// TwinCAT 3 PLC project PLC_TMO_VAC
// ProgramVersion: 3.1.4022.7
// libraries:
//   LCLS General, * (SLAC)
//   LCLS Vacuum, * (SLAC - LCLS)
//   LCLSVacuumSerialDriverLib, * (SLAC - LCLS)
//   PMPS, * (SLAC - LCLS)
//   Tc2_SerialCom, * (Beckhoff Automation GmbH)
//   Tc2_Standard, * (Beckhoff Automation GmbH)
//   Tc2_System, * (Beckhoff Automation GmbH)
//   Tc3_Module, * (Beckhoff Automation GmbH)
// project tree:
//   / ComTask.TcTTO (not stored), FSVTask.TcTTO (not stored), PlcTask.TcTTO (not stored)
//   GVLs/ GVL_COM.TcGVL (not stored), GVL_FEE_Device.TcGVL, GVL_FSV_PMPS.TcGVL, GVL_FS_Devices.TcGVL, GVL_Hutch_Gauges.TcGVL, GVL_Hutch_Pumps.TcGVL (not stored), GVL_Hutch_Valves.TcGVL (not stored), GVL_PMPS.TcGVL, GVL_Variables.TcGVL
//   POUs/ DIAGNOSTICS.TcPOU, F_Turbo_Protection_ILK.TcPOU (not stored), MAIN.TcPOU, PMPS.TcPOU, PRG_COM.TcPOU (not stored), PRG_FEE.TcPOU, PRG_FSV.TcPOU, PRG_FSV_Interfaces.TcPOU (not stored), PRG_Hutch_Beamline_Valves.TcPOU (not stored), PRG_Hutch_Gauges.TcPOU (not stored), PRG_Roughing_Pumps.TcPOU, PRG_Section_2.TcPOU (not stored)
// real-time tasks:
//   TASK PlcTask: cycle T#10ms, priority 20, ADS port 350
//   TASK ComTask: cycle T#11ms, priority 1, ADS port 351
//   TASK FSVTask: cycle T#2ms, priority 2, ADS port 352
// I/O:
//   DEVICE Device 1 (EtherCAT), AmsNetId 172.21.132.22.2.1
//     B940-R20-CX0 (EK1200) [EK1200-5000 EtherCAT Power supply (2A E-Bus)]
//       CX0_E1 (EL2202)
//       CX0_E2_EXILK (EL1008)
//       CX0_E3 (EL2008)
//       CX0_E4 (EL2794)
//       CX0_E5 (EL6070)
//       CX0_E6_QPC1 (EL3064)
//       CX0_E7_QPC1 (EL1004)
//       CX0_E8_QPC1 (EL2794)
//       CX0_E9_QPC2 (EL3064)
//       CX0_E10_QPC2 (EL1004)
//       CX0_E11_QPC2 (EL2794)
//       CX0_E12 (EL6001)
//       EK1122-0080
//       PMPS_PRE
//       CX0_EK1110
//     B940_R20_EK0 (EK1100) [EK1100 EtherCAT Coupler (2A E-Bus)]
//       R20_EK0_E1 (EL3064)
//       R20_EK0_E2 (EL3064)
//       R20_EK0_E3 (EL2794)
//       R20_EK0_E4 (EL9505)
//       R20_EK0_E5 (EL1124)
//       R20_EK0_E6 (EK1110)
//     B940_K4S20_EK0  (EK1100)
//     B940_K4S20_EB1  (EP2338-0002)
//     B940_K4S20_EB2  (EP3174-0002)
//     B940_K4S20_EB3 (EP2624-0002)
//     B940_K4S24_EB1 (EP3174-0002)
//     B940_K4S24_EB2 (EP2624-0002)
//     B940_K4S28_EB1 (EP3174-0002)
//     B940_K4S28_EB2 (EP2624-0002)
//     B940_K4S33_EB1 (EP2338-0002)
//     B940_K4S33_EB2 (EP3174-0002)
//     B940_K4S33_EB3 (EP2624-0002)
//     TMO_WALL_WEST_EP01 (EP4374-0002)
//     TMO_K4S2_DRL_01 (EK1100)
//     TMO_K4S2_DRL_02 (EK1100)
//     TMO_K4S2_ EP1 (EP4374-0002)
//     TMO_K4S6_ EP1 (EP4374-0002)
//     TMO_K4S6_DRL_01 (EK1100)
//     TMO_K4S8_DRL_01 (EK1100)
// variable links:
//   PLC_TMO_VAC Instance <-> Device 1 (EtherCAT)/B940-R20-CX0 (EK1200)/CX0_E1 (EL2202)
//     PlcTask Outputs/GVL_PMPS.g_FastFaultOutput1.q_xFastFaultOut <-> Channel 1/Output
//     PlcTask Outputs/GVL_PMPS.g_FastFaultOutput2.q_xFastFaultOut <-> Channel 2/Output
//   PLC_TMO_VAC Instance <-> Device 1 (EtherCAT)/B940-R20-CX0 (EK1200)/CX0_E10_QPC2 (EL1004)
//     PlcTask Inputs/GVL_FEE_Device.PC4K4_XTES_PIP_01.i_xSP_DI <-> Channel 1/Input
//     PlcTask Inputs/GVL_Hutch_Pumps.MR2K4_KBO_PIP_01.i_xSP_DI <-> Channel 2/Input
//     PlcTask Inputs/GVL_Hutch_Pumps.MR4K4_KBO_PIP_01.i_xSP_DI <-> Channel 4/Input
//     PlcTask Inputs/GVL_Hutch_Pumps.PA2K4_IP1_PIP_01.i_xSP_DI <-> Channel 3/Input
//   PLC_TMO_VAC Instance <-> Device 1 (EtherCAT)/B940-R20-CX0 (EK1200)/CX0_E11_QPC2 (EL2794)
//     PlcTask Outputs/GVL_FEE_Device.PC4K4_XTES_PIP_01.q_xHVEna_DO <-> Channel 1/Output
//     PlcTask Outputs/GVL_Hutch_Pumps.MR2K4_KBO_PIP_01.q_xHVEna_DO <-> Channel 2/Output
//     PlcTask Outputs/GVL_Hutch_Pumps.MR4K4_KBO_PIP_01.q_xHVEna_DO <-> Channel 4/Output
//     PlcTask Outputs/GVL_Hutch_Pumps.PA2K4_IP1_PIP_01.q_xHVEna_DO <-> Channel 3/Output
//   PLC_TMO_VAC Instance <-> Device 1 (EtherCAT)/B940-R20-CX0 (EK1200)/CX0_E2_EXILK (EL1008)
//     PlcTask Inputs/GVL_FEE_Device.USVacOk_HI <-> Channel 1/Input
//     PlcTask Inputs/GVL_FEE_Device.USVacOk_LO <-> Channel 3/Input
//   PLC_TMO_VAC Instance <-> Device 1 (EtherCAT)/B940-R20-CX0 (EK1200)/CX0_E6_QPC1 (EL3064)
//     PlcTask Inputs/GVL_FEE_Device.MR1K4_SOMS_PIP_01.i_iPRESS <-> AI Standard Channel 1/Value
//     PlcTask Inputs/GVL_FEE_Device.ST1K4_TEST_PIP_01.i_iPRESS <-> AI Standard Channel 2/Value
//     PlcTask Inputs/GVL_FEE_Device.ST2K4_BCS_PIP_01.i_iPRESS <-> AI Standard Channel 3/Value
//     PlcTask Inputs/GVL_FEE_Device.ST3K4_PPS_PIP_01.i_iPRESS <-> AI Standard Channel 4/Value
//   PLC_TMO_VAC Instance <-> Device 1 (EtherCAT)/B940-R20-CX0 (EK1200)/CX0_E7_QPC1 (EL1004)
//     PlcTask Inputs/GVL_FEE_Device.MR1K4_SOMS_PIP_01.i_xSP_DI <-> Channel 1/Input
//     PlcTask Inputs/GVL_FEE_Device.ST1K4_TEST_PIP_01.i_xSP_DI <-> Channel 2/Input
//     PlcTask Inputs/GVL_FEE_Device.ST2K4_BCS_PIP_01.i_xSP_DI <-> Channel 3/Input
//     PlcTask Inputs/GVL_FEE_Device.ST3K4_PPS_PIP_01.i_xSP_DI <-> Channel 4/Input
//   PLC_TMO_VAC Instance <-> Device 1 (EtherCAT)/B940-R20-CX0 (EK1200)/CX0_E8_QPC1 (EL2794)
//     PlcTask Outputs/GVL_FEE_Device.MR1K4_SOMS_PIP_01.q_xHVEna_DO <-> Channel 1/Output
//     PlcTask Outputs/GVL_FEE_Device.ST1K4_TEST_PIP_01.q_xHVEna_DO <-> Channel 2/Output
//     PlcTask Outputs/GVL_FEE_Device.ST2K4_BCS_PIP_01.q_xHVEna_DO <-> Channel 3/Output
//     PlcTask Outputs/GVL_FEE_Device.ST3K4_PPS_PIP_01.q_xHVEna_DO <-> Channel 4/Output
//   PLC_TMO_VAC Instance <-> Device 1 (EtherCAT)/B940-R20-CX0 (EK1200)/CX0_E9_QPC2 (EL3064)
//     PlcTask Inputs/GVL_FEE_Device.PC4K4_XTES_PIP_01.i_iPRESS <-> AI Standard Channel 1/Value
//     PlcTask Inputs/GVL_Hutch_Pumps.MR2K4_KBO_PIP_01.i_iPRESS <-> AI Standard Channel 2/Value
//     PlcTask Inputs/GVL_Hutch_Pumps.MR4K4_KBO_PIP_01.i_iPRESS <-> AI Standard Channel 4/Value
//     PlcTask Inputs/GVL_Hutch_Pumps.PA2K4_IP1_PIP_01.i_iPRESS <-> AI Standard Channel 3/Value
//   PLC_TMO_VAC Instance <-> Device 1 (EtherCAT)/B940-R20-CX0 (EK1200)/PMPS_PRE
//     PlcTask Inputs/PMPS.fbArbiterIO.i_stCurrentBP <-> IO Inputs/CurrentBP
//     PlcTask Inputs/PMPS.fbArbiterIO.xTxPDO_state <-> SYNC Inputs/TxPDO state
//     PlcTask Inputs/PMPS.fbArbiterIO.xTxPDO_toggle <-> SYNC Inputs/TxPDO toggle
//     PlcTask Outputs/PMPS.fbArbiterIO.q_stRequestedBP <-> IO Outputs/RequestedBP
//   PLC_TMO_VAC Instance <-> Device 1 (EtherCAT)/B940_K4S20_EB1  (EP2338-0002)
//     PlcTask Inputs/GVL_FEE_Device.TV1K4_VGC_01.i_xClsLS <-> Channel 2/Input
//     PlcTask Inputs/GVL_FEE_Device.TV1K4_VGC_02.i_xClsLS <-> Channel 6/Input
//     PlcTask Inputs/GVL_FEE_Device.TV1K4_VGC_01.i_xOpnLS <-> Channel 1/Input
//     PlcTask Inputs/GVL_FEE_Device.TV1K4_VGC_02.i_xOpnLS <-> Channel 5/Input
//     PlcTask Outputs/GVL_FEE_Device.TV1K4_VGC_01.q_xOPN_DO <-> Channel 11/Output
//     PlcTask Outputs/GVL_FEE_Device.TV1K4_VGC_02.q_xOPN_DO <-> Channel 15/Output
//   PLC_TMO_VAC Instance <-> Device 1 (EtherCAT)/B940_K4S20_EB2  (EP3174-0002)
//     PlcTask Inputs/GVL_FEE_Device.TV1K4_GCC_01.i_iPRESS_R <-> AI Standard Channel 2/Value
//     PlcTask Inputs/GVL_FEE_Device.TV1K4_GPI_01.i_iPRESS_R <-> AI Standard Channel 1/Value
//   PLC_TMO_VAC Instance <-> Device 1 (EtherCAT)/B940_K4S20_EB3 (EP2624-0002)
//     PlcTask Outputs/GVL_FEE_Device.TV1K4_GCC_01.q_xHV_DIS <-> Channel 1/Output
//   PLC_TMO_VAC Instance <-> Device 1 (EtherCAT)/B940_K4S24_EB1 (EP3174-0002)
//     PlcTask Inputs/GVL_FEE_Device.ST1K4_TEST_GCC_01.i_iPRESS_R <-> AI Standard Channel 2/Value
//     PlcTask Inputs/GVL_FEE_Device.ST1K4_TEST_GPI_01.i_iPRESS_R <-> AI Standard Channel 1/Value
//   PLC_TMO_VAC Instance <-> Device 1 (EtherCAT)/B940_K4S24_EB2 (EP2624-0002)
//     PlcTask Outputs/GVL_FEE_Device.ST1K4_TEST_GCC_01.q_xHV_DIS <-> Channel 1/Output
//   PLC_TMO_VAC Instance <-> Device 1 (EtherCAT)/B940_K4S28_EB1 (EP3174-0002)
//     PlcTask Inputs/GVL_FEE_Device.ST2K4_BCS_GCC_01.i_iPRESS_R <-> AI Standard Channel 2/Value
//     PlcTask Inputs/GVL_FEE_Device.ST2K4_BCS_GPI_01.i_iPRESS_R <-> AI Standard Channel 1/Value
//   PLC_TMO_VAC Instance <-> Device 1 (EtherCAT)/B940_K4S28_EB2 (EP2624-0002)
//     PlcTask Outputs/GVL_FEE_Device.ST2K4_BCS_GCC_01.q_xHV_DIS <-> Channel 1/Output
//   PLC_TMO_VAC Instance <-> Device 1 (EtherCAT)/B940_K4S33_EB1 (EP2338-0002)
//     PlcTask Inputs/GVL_FEE_Device.ST3K4_PPS_VGC_01.i_xClsLS <-> Channel 2/Input
//     PlcTask Inputs/GVL_FEE_Device.ST3K4_PPS_VGC_01.i_xOpnLS <-> Channel 1/Input
//     PlcTask Outputs/GVL_FEE_Device.ST3K4_PPS_VGC_01.q_xOPN_DO <-> Channel 11/Output
//   PLC_TMO_VAC Instance <-> Device 1 (EtherCAT)/B940_K4S33_EB2 (EP3174-0002)
//     PlcTask Inputs/GVL_FEE_Device.PC4K4_XTES_GCC_01.i_iPRESS_R <-> AI Standard Channel 2/Value
//     PlcTask Inputs/GVL_FEE_Device.PC4K4_XTES_GPI_01.i_iPRESS_R <-> AI Standard Channel 1/Value
//   PLC_TMO_VAC Instance <-> Device 1 (EtherCAT)/B940_K4S33_EB3 (EP2624-0002)
//     PlcTask Outputs/GVL_FEE_Device.PC4K4_XTES_GCC_01.q_xHV_DIS <-> Channel 1/Output
//   PLC_TMO_VAC Instance <-> Device 1 (EtherCAT)/B940_R20_EK0 (EK1100)/R20_EK0_E5_MKS937B (EL1124)
//     FSVTask Inputs/GVL_FS_Devices.MR3K4_KBO_VFS_1.i_xTrigger <-> Channel 1/Input
//     FSVTask Inputs/GVL_FS_Devices.MR4K4_KBO_VFS_1.i_xTrigger <-> Channel 1/Input
//     FSVTask Inputs/GVL_FS_Devices.TV1K4_VFS_1.i_xTrigger <-> Channel 1/Input
//   PLC_TMO_VAC Instance <-> Device 1 (EtherCAT)/TMO_K4S2_ EP1 (EP4374-0002)
//     PlcTask Inputs/GVL_Hutch_Gauges.TMO_ROUGH1_GPI_02.i_iPRESS_R <-> AI Inputs Channel 1/Value
//     PlcTask Inputs/GVL_Hutch_Gauges.TMO_ROUGH2_GPI_02.i_iPRESS_R <-> AI Inputs Channel 2/Value
//     PlcTask Outputs/GVL_Hutch_Valves.TMO_ROUGH1_VFV_02.q_iRawPosition <-> AO Outputs Channel 3/Analog output
//     PlcTask Outputs/GVL_Hutch_Valves.TMO_ROUGH2_VFV_01.q_iRawPosition <-> AO Outputs Channel 4/Analog output
//   PLC_TMO_VAC Instance <-> Device 1 (EtherCAT)/TMO_K4S2_DRL_01 (EK1100)/K4S2_01_E1_VFS (EL1004)
//     FSVTask Inputs/GVL_FS_Devices.MR3K4_KBO_VFS_1.i_xClsLS <-> Channel 1/Input
//     FSVTask Inputs/GVL_FS_Devices.MR3K4_KBO_VFS_1.i_xOpnLS <-> Channel 2/Input
//   PLC_TMO_VAC Instance <-> Device 1 (EtherCAT)/TMO_K4S2_DRL_01 (EK1100)/K4S2_01_E3_VFS (EL2202)
//     FSVTask Outputs/GVL_FS_Devices.MR3K4_KBO_VFS_1.q_xClose_A <-> Channel 1/Output
//     FSVTask Outputs/GVL_FS_Devices.MR3K4_KBO_VFS_1.q_xClose_B <-> Channel 2/Output
//   PLC_TMO_VAC Instance <-> Device 1 (EtherCAT)/TMO_K4S2_DRL_01 (EK1100)/K4S2_01_E4_VFS (EL2202)
//     FSVTask Outputs/GVL_FS_Devices.MR3K4_KBO_VFS_1.q_xClose_C <-> Channel 1/Output
//     FSVTask Outputs/GVL_FS_Devices.MR3K4_KBO_VFS_1.q_xOPN_DO <-> Channel 2/Output
//   PLC_TMO_VAC Instance <-> Device 1 (EtherCAT)/TMO_K4S2_DRL_01 (EK1100)/K4S2_01_E5 (EL1004)
//     PlcTask Inputs/GVL_Hutch_Valves.MR2K4_KBO_VWC_01.i_xClsLS <-> Channel 2/Input
//     PlcTask Inputs/GVL_Hutch_Valves.MR3K4_KBO_VWC_01.i_xClsLS <-> Channel 4/Input
//     PlcTask Inputs/GVL_Hutch_Valves.MR2K4_KBO_VWC_01.i_xOpnLS <-> Channel 1/Input
//     PlcTask Inputs/GVL_Hutch_Valves.MR3K4_KBO_VWC_01.i_xOpnLS <-> Channel 3/Input
//   PLC_TMO_VAC Instance <-> Device 1 (EtherCAT)/TMO_K4S2_DRL_01 (EK1100)/K4S2_01_E6 (EL2004)
//     PlcTask Outputs/GVL_Hutch_Valves.MR2K4_KBO_VWC_01.q_xOPN_DO <-> Channel 1/Output
//     PlcTask Outputs/GVL_Hutch_Valves.MR3K4_KBO_VWC_01.q_xOPN_DO <-> Channel 2/Output
//   PLC_TMO_VAC Instance <-> Device 1 (EtherCAT)/TMO_K4S2_DRL_02 (EK1100)/K4S2_02_E1 (EL3174)
//     PlcTask Inputs/GVL_Hutch_Gauges.MR2K4_KBO_GCC_01.i_iPRESS_R <-> AI Standard Channel 3/Value
//     PlcTask Inputs/GVL_Hutch_Gauges.MR2K4_KBO_GPI_01.i_iPRESS_R <-> AI Standard Channel 2/Value
//     PlcTask Inputs/GVL_Hutch_Gauges.PA1K4_IP1_GCC_01.i_iPRESS_R <-> AI Standard Channel 4/Value
//   PLC_TMO_VAC Instance <-> Device 1 (EtherCAT)/TMO_K4S2_DRL_02 (EK1100)/K4S2_02_E10 (EL6021)
//     ComTask Inputs/GVL_COM.K4S2_02_E10_stComIn/D[0] <-> COM TxPDO-Map Inputs/Data In 0
//     ComTask Inputs/GVL_COM.K4S2_02_E10_stComIn/D[10] <-> COM TxPDO-Map Inputs/Data In 10
//     ComTask Inputs/GVL_COM.K4S2_02_E10_stComIn/D[11] <-> COM TxPDO-Map Inputs/Data In 11
//     ComTask Inputs/GVL_COM.K4S2_02_E10_stComIn/D[12] <-> COM TxPDO-Map Inputs/Data In 12
//     ComTask Inputs/GVL_COM.K4S2_02_E10_stComIn/D[13] <-> COM TxPDO-Map Inputs/Data In 13
//     ComTask Inputs/GVL_COM.K4S2_02_E10_stComIn/D[14] <-> COM TxPDO-Map Inputs/Data In 14
//     ComTask Inputs/GVL_COM.K4S2_02_E10_stComIn/D[15] <-> COM TxPDO-Map Inputs/Data In 15
//     ComTask Inputs/GVL_COM.K4S2_02_E10_stComIn/D[16] <-> COM TxPDO-Map Inputs/Data In 16
//     ComTask Inputs/GVL_COM.K4S2_02_E10_stComIn/D[17] <-> COM TxPDO-Map Inputs/Data In 17
//     ComTask Inputs/GVL_COM.K4S2_02_E10_stComIn/D[18] <-> COM TxPDO-Map Inputs/Data In 18
//     ComTask Inputs/GVL_COM.K4S2_02_E10_stComIn/D[19] <-> COM TxPDO-Map Inputs/Data In 19
//     ComTask Inputs/GVL_COM.K4S2_02_E10_stComIn/D[1] <-> COM TxPDO-Map Inputs/Data In 1
//     ComTask Inputs/GVL_COM.K4S2_02_E10_stComIn/D[20] <-> COM TxPDO-Map Inputs/Data In 20
//     ComTask Inputs/GVL_COM.K4S2_02_E10_stComIn/D[21] <-> COM TxPDO-Map Inputs/Data In 21
//     ComTask Inputs/GVL_COM.K4S2_02_E10_stComIn/D[2] <-> COM TxPDO-Map Inputs/Data In 2
//     ComTask Inputs/GVL_COM.K4S2_02_E10_stComIn/D[3] <-> COM TxPDO-Map Inputs/Data In 3
//     ComTask Inputs/GVL_COM.K4S2_02_E10_stComIn/D[4] <-> COM TxPDO-Map Inputs/Data In 4
//     ComTask Inputs/GVL_COM.K4S2_02_E10_stComIn/D[5] <-> COM TxPDO-Map Inputs/Data In 5
//     ComTask Inputs/GVL_COM.K4S2_02_E10_stComIn/D[6] <-> COM TxPDO-Map Inputs/Data In 6
//     ComTask Inputs/GVL_COM.K4S2_02_E10_stComIn/D[7] <-> COM TxPDO-Map Inputs/Data In 7
//     ComTask Inputs/GVL_COM.K4S2_02_E10_stComIn/D[8] <-> COM TxPDO-Map Inputs/Data In 8
//     ComTask Inputs/GVL_COM.K4S2_02_E10_stComIn/D[9] <-> COM TxPDO-Map Inputs/Data In 9
//     ComTask Inputs/GVL_COM.K4S2_02_E10_stComIn/Status <-> COM TxPDO-Map Inputs/Status
//     ComTask Outputs/GVL_COM.K4S2_02_E10_stComOut/Ctrl <-> COM RxPDO-Map Outputs/Ctrl
//     ComTask Outputs/GVL_COM.K4S2_02_E10_stComOut/D[0] <-> COM RxPDO-Map Outputs/Data Out 0
//     ComTask Outputs/GVL_COM.K4S2_02_E10_stComOut/D[10] <-> COM RxPDO-Map Outputs/Data Out 10
//     ComTask Outputs/GVL_COM.K4S2_02_E10_stComOut/D[11] <-> COM RxPDO-Map Outputs/Data Out 11
//     ComTask Outputs/GVL_COM.K4S2_02_E10_stComOut/D[12] <-> COM RxPDO-Map Outputs/Data Out 12
//     ComTask Outputs/GVL_COM.K4S2_02_E10_stComOut/D[13] <-> COM RxPDO-Map Outputs/Data Out 13
//     ComTask Outputs/GVL_COM.K4S2_02_E10_stComOut/D[14] <-> COM RxPDO-Map Outputs/Data Out 14
//     ComTask Outputs/GVL_COM.K4S2_02_E10_stComOut/D[15] <-> COM RxPDO-Map Outputs/Data Out 15
//     ComTask Outputs/GVL_COM.K4S2_02_E10_stComOut/D[16] <-> COM RxPDO-Map Outputs/Data Out 16
//     ComTask Outputs/GVL_COM.K4S2_02_E10_stComOut/D[17] <-> COM RxPDO-Map Outputs/Data Out 17
//     ComTask Outputs/GVL_COM.K4S2_02_E10_stComOut/D[18] <-> COM RxPDO-Map Outputs/Data Out 18
//     ComTask Outputs/GVL_COM.K4S2_02_E10_stComOut/D[19] <-> COM RxPDO-Map Outputs/Data Out 19
//     ComTask Outputs/GVL_COM.K4S2_02_E10_stComOut/D[1] <-> COM RxPDO-Map Outputs/Data Out 1
//     ComTask Outputs/GVL_COM.K4S2_02_E10_stComOut/D[20] <-> COM RxPDO-Map Outputs/Data Out 20
//     ComTask Outputs/GVL_COM.K4S2_02_E10_stComOut/D[21] <-> COM RxPDO-Map Outputs/Data Out 21
//     ComTask Outputs/GVL_COM.K4S2_02_E10_stComOut/D[2] <-> COM RxPDO-Map Outputs/Data Out 2
//     ComTask Outputs/GVL_COM.K4S2_02_E10_stComOut/D[3] <-> COM RxPDO-Map Outputs/Data Out 3
//     ComTask Outputs/GVL_COM.K4S2_02_E10_stComOut/D[4] <-> COM RxPDO-Map Outputs/Data Out 4
//     ComTask Outputs/GVL_COM.K4S2_02_E10_stComOut/D[5] <-> COM RxPDO-Map Outputs/Data Out 5
//     ComTask Outputs/GVL_COM.K4S2_02_E10_stComOut/D[6] <-> COM RxPDO-Map Outputs/Data Out 6
//     ComTask Outputs/GVL_COM.K4S2_02_E10_stComOut/D[7] <-> COM RxPDO-Map Outputs/Data Out 7
//     ComTask Outputs/GVL_COM.K4S2_02_E10_stComOut/D[8] <-> COM RxPDO-Map Outputs/Data Out 8
//     ComTask Outputs/GVL_COM.K4S2_02_E10_stComOut/D[9] <-> COM RxPDO-Map Outputs/Data Out 9
//   PLC_TMO_VAC Instance <-> Device 1 (EtherCAT)/TMO_K4S2_DRL_02 (EK1100)/K4S2_02_E11 (EL1004)
//     PlcTask Inputs/GVL_Hutch_Pumps.PA1K4_IP1_PTM_01.i_xAtSpd <-> Channel 2/Input
//     PlcTask Inputs/GVL_Hutch_Pumps.PA1K4_IP1_PTM_02.i_xAtSpd <-> Channel 4/Input
//     PlcTask Inputs/GVL_Hutch_Pumps.PA1K4_IP1_PTM_01.i_xFaultNC <-> Channel 1/Input
//     PlcTask Inputs/GVL_Hutch_Pumps.PA1K4_IP1_PTM_02.i_xFaultNC <-> Channel 3/Input
//   PLC_TMO_VAC Instance <-> Device 1 (EtherCAT)/TMO_K4S2_DRL_02 (EK1100)/K4S2_02_E12 (EL2794)
//     PlcTask Outputs/GVL_Hutch_Pumps.PA1K4_IP1_PTM_01.q_RunDO <-> Channel 1/Output
//     PlcTask Outputs/GVL_Hutch_Pumps.PA1K4_IP1_PTM_02.q_RunDO <-> Channel 3/Output
//     PlcTask Outputs/GVL_Hutch_Pumps.PA1K4_IP1_PTM_01.q_xReset <-> Channel 2/Output
//     PlcTask Outputs/GVL_Hutch_Pumps.PA1K4_IP1_PTM_02.q_xReset <-> Channel 4/Output
//   PLC_TMO_VAC Instance <-> Device 1 (EtherCAT)/TMO_K4S2_DRL_02 (EK1100)/K4S2_02_E13 (EL1004)
//     PlcTask Inputs/GVL_Hutch_Pumps.PA1K4_IP1_PTM_03.i_xAtSpd <-> Channel 2/Input
//     PlcTask Inputs/GVL_Hutch_Pumps.PA1K4_IP1_PTM_03.i_xFaultNC <-> Channel 1/Input
//   PLC_TMO_VAC Instance <-> Device 1 (EtherCAT)/TMO_K4S2_DRL_02 (EK1100)/K4S2_02_E14 (EL2794)
//     PlcTask Outputs/GVL_Hutch_Pumps.PA1K4_IP1_PTM_03.q_RunDO <-> Channel 1/Output
//     PlcTask Outputs/GVL_Hutch_Pumps.PA1K4_IP1_PTM_03.q_xReset <-> Channel 2/Output
//   PLC_TMO_VAC Instance <-> Device 1 (EtherCAT)/TMO_K4S2_DRL_02 (EK1100)/K4S2_02_E15 (EL1004)
//     PlcTask Inputs/GVL_Hutch_Pumps.IM4K4_PPM_PTM_01.i_xAtSpd <-> Channel 2/Input
//     PlcTask Inputs/GVL_Hutch_Pumps.IM4K4_PPM_PTM_01.i_xFaultNC <-> Channel 1/Input
//     PlcTask Inputs/GVL_Hutch_Pumps.LI1K4_IP1_PTM_01.i_xAtSpd <-> Channel 4/Input
//     PlcTask Inputs/GVL_Hutch_Pumps.LI1K4_IP1_PTM_01.i_xFaultNC <-> Channel 3/Input
//   PLC_TMO_VAC Instance <-> Device 1 (EtherCAT)/TMO_K4S2_DRL_02 (EK1100)/K4S2_02_E16 (EL2794)
//     PlcTask Outputs/GVL_Hutch_Pumps.IM4K4_PPM_PTM_01.q_RunDO <-> Channel 1/Output
//     PlcTask Outputs/GVL_Hutch_Pumps.LI1K4_IP1_PTM_01.q_RunDO <-> Channel 2/Output
//   PLC_TMO_VAC Instance <-> Device 1 (EtherCAT)/TMO_K4S2_DRL_02 (EK1100)/K4S2_02_E17 (EL6001)
//     ComTask Inputs/GVL_COM.K4S2_02_E17_stComIn/D[0] <-> COM Inputs/Data In 0
//     ComTask Inputs/GVL_COM.K4S2_02_E17_stComIn/D[10] <-> COM Inputs/Data In 10
//     ComTask Inputs/GVL_COM.K4S2_02_E17_stComIn/D[11] <-> COM Inputs/Data In 11
//     ComTask Inputs/GVL_COM.K4S2_02_E17_stComIn/D[12] <-> COM Inputs/Data In 12
//     ComTask Inputs/GVL_COM.K4S2_02_E17_stComIn/D[13] <-> COM Inputs/Data In 13
//     ComTask Inputs/GVL_COM.K4S2_02_E17_stComIn/D[14] <-> COM Inputs/Data In 14
//     ComTask Inputs/GVL_COM.K4S2_02_E17_stComIn/D[15] <-> COM Inputs/Data In 15
//     ComTask Inputs/GVL_COM.K4S2_02_E17_stComIn/D[16] <-> COM Inputs/Data In 16
//     ComTask Inputs/GVL_COM.K4S2_02_E17_stComIn/D[17] <-> COM Inputs/Data In 17
//     ComTask Inputs/GVL_COM.K4S2_02_E17_stComIn/D[18] <-> COM Inputs/Data In 18
//     ComTask Inputs/GVL_COM.K4S2_02_E17_stComIn/D[19] <-> COM Inputs/Data In 19
//     ComTask Inputs/GVL_COM.K4S2_02_E17_stComIn/D[1] <-> COM Inputs/Data In 1
//     ComTask Inputs/GVL_COM.K4S2_02_E17_stComIn/D[20] <-> COM Inputs/Data In 20
//     ComTask Inputs/GVL_COM.K4S2_02_E17_stComIn/D[21] <-> COM Inputs/Data In 21
//     ComTask Inputs/GVL_COM.K4S2_02_E17_stComIn/D[2] <-> COM Inputs/Data In 2
//     ComTask Inputs/GVL_COM.K4S2_02_E17_stComIn/D[3] <-> COM Inputs/Data In 3
//     ComTask Inputs/GVL_COM.K4S2_02_E17_stComIn/D[4] <-> COM Inputs/Data In 4
//     ComTask Inputs/GVL_COM.K4S2_02_E17_stComIn/D[5] <-> COM Inputs/Data In 5
//     ComTask Inputs/GVL_COM.K4S2_02_E17_stComIn/D[6] <-> COM Inputs/Data In 6
//     ComTask Inputs/GVL_COM.K4S2_02_E17_stComIn/D[7] <-> COM Inputs/Data In 7
//     ComTask Inputs/GVL_COM.K4S2_02_E17_stComIn/D[8] <-> COM Inputs/Data In 8
//     ComTask Inputs/GVL_COM.K4S2_02_E17_stComIn/D[9] <-> COM Inputs/Data In 9
//     ComTask Inputs/GVL_COM.K4S2_02_E17_stComIn/Status <-> COM Inputs/Status
//     ComTask Outputs/GVL_COM.K4S2_02_E17_stComOut/Ctrl <-> COM Outputs/Ctrl
//     ComTask Outputs/GVL_COM.K4S2_02_E17_stComOut/D[0] <-> COM Outputs/Data Out 0
//     ComTask Outputs/GVL_COM.K4S2_02_E17_stComOut/D[10] <-> COM Outputs/Data Out 10
//     ComTask Outputs/GVL_COM.K4S2_02_E17_stComOut/D[11] <-> COM Outputs/Data Out 11
//     ComTask Outputs/GVL_COM.K4S2_02_E17_stComOut/D[12] <-> COM Outputs/Data Out 12
//     ComTask Outputs/GVL_COM.K4S2_02_E17_stComOut/D[13] <-> COM Outputs/Data Out 13
//     ComTask Outputs/GVL_COM.K4S2_02_E17_stComOut/D[14] <-> COM Outputs/Data Out 14
//     ComTask Outputs/GVL_COM.K4S2_02_E17_stComOut/D[15] <-> COM Outputs/Data Out 15
//     ComTask Outputs/GVL_COM.K4S2_02_E17_stComOut/D[16] <-> COM Outputs/Data Out 16
//     ComTask Outputs/GVL_COM.K4S2_02_E17_stComOut/D[17] <-> COM Outputs/Data Out 17
//     ComTask Outputs/GVL_COM.K4S2_02_E17_stComOut/D[18] <-> COM Outputs/Data Out 18
//     ComTask Outputs/GVL_COM.K4S2_02_E17_stComOut/D[19] <-> COM Outputs/Data Out 19
//     ComTask Outputs/GVL_COM.K4S2_02_E17_stComOut/D[1] <-> COM Outputs/Data Out 1
//     ComTask Outputs/GVL_COM.K4S2_02_E17_stComOut/D[20] <-> COM Outputs/Data Out 20
//     ComTask Outputs/GVL_COM.K4S2_02_E17_stComOut/D[21] <-> COM Outputs/Data Out 21
//     ComTask Outputs/GVL_COM.K4S2_02_E17_stComOut/D[2] <-> COM Outputs/Data Out 2
//     ComTask Outputs/GVL_COM.K4S2_02_E17_stComOut/D[3] <-> COM Outputs/Data Out 3
//     ComTask Outputs/GVL_COM.K4S2_02_E17_stComOut/D[4] <-> COM Outputs/Data Out 4
//     ComTask Outputs/GVL_COM.K4S2_02_E17_stComOut/D[5] <-> COM Outputs/Data Out 5
//     ComTask Outputs/GVL_COM.K4S2_02_E17_stComOut/D[6] <-> COM Outputs/Data Out 6
//     ComTask Outputs/GVL_COM.K4S2_02_E17_stComOut/D[7] <-> COM Outputs/Data Out 7
//     ComTask Outputs/GVL_COM.K4S2_02_E17_stComOut/D[8] <-> COM Outputs/Data Out 8
//     ComTask Outputs/GVL_COM.K4S2_02_E17_stComOut/D[9] <-> COM Outputs/Data Out 9
//   PLC_TMO_VAC Instance <-> Device 1 (EtherCAT)/TMO_K4S2_DRL_02 (EK1100)/K4S2_02_E18 (EL6001)
//     ComTask Inputs/GVL_COM.K4S2_02_E18_stComIn/D[0] <-> COM Inputs/Data In 0
//     ComTask Inputs/GVL_COM.K4S2_02_E18_stComIn/D[10] <-> COM Inputs/Data In 10
//     ComTask Inputs/GVL_COM.K4S2_02_E18_stComIn/D[11] <-> COM Inputs/Data In 11
//     ComTask Inputs/GVL_COM.K4S2_02_E18_stComIn/D[12] <-> COM Inputs/Data In 12
//     ComTask Inputs/GVL_COM.K4S2_02_E18_stComIn/D[13] <-> COM Inputs/Data In 13
//     ComTask Inputs/GVL_COM.K4S2_02_E18_stComIn/D[14] <-> COM Inputs/Data In 14
//     ComTask Inputs/GVL_COM.K4S2_02_E18_stComIn/D[15] <-> COM Inputs/Data In 15
//     ComTask Inputs/GVL_COM.K4S2_02_E18_stComIn/D[16] <-> COM Inputs/Data In 16
//     ComTask Inputs/GVL_COM.K4S2_02_E18_stComIn/D[17] <-> COM Inputs/Data In 17
//     ComTask Inputs/GVL_COM.K4S2_02_E18_stComIn/D[18] <-> COM Inputs/Data In 18
//     ComTask Inputs/GVL_COM.K4S2_02_E18_stComIn/D[19] <-> COM Inputs/Data In 19
//     ComTask Inputs/GVL_COM.K4S2_02_E18_stComIn/D[1] <-> COM Inputs/Data In 1
//     ComTask Inputs/GVL_COM.K4S2_02_E18_stComIn/D[20] <-> COM Inputs/Data In 20
//     ComTask Inputs/GVL_COM.K4S2_02_E18_stComIn/D[21] <-> COM Inputs/Data In 21
//     ComTask Inputs/GVL_COM.K4S2_02_E18_stComIn/D[2] <-> COM Inputs/Data In 2
//     ComTask Inputs/GVL_COM.K4S2_02_E18_stComIn/D[3] <-> COM Inputs/Data In 3
//     ComTask Inputs/GVL_COM.K4S2_02_E18_stComIn/D[4] <-> COM Inputs/Data In 4
//     ComTask Inputs/GVL_COM.K4S2_02_E18_stComIn/D[5] <-> COM Inputs/Data In 5
//     ComTask Inputs/GVL_COM.K4S2_02_E18_stComIn/D[6] <-> COM Inputs/Data In 6
//     ComTask Inputs/GVL_COM.K4S2_02_E18_stComIn/D[7] <-> COM Inputs/Data In 7
//     ComTask Inputs/GVL_COM.K4S2_02_E18_stComIn/D[8] <-> COM Inputs/Data In 8
//     ComTask Inputs/GVL_COM.K4S2_02_E18_stComIn/D[9] <-> COM Inputs/Data In 9
//     ComTask Inputs/GVL_COM.K4S2_02_E18_stComIn/Status <-> COM Inputs/Status
//     ComTask Outputs/GVL_COM.K4S2_02_E18_stComOut/Ctrl <-> COM Outputs/Ctrl
//     ComTask Outputs/GVL_COM.K4S2_02_E18_stComOut/D[0] <-> COM Outputs/Data Out 0
//     ComTask Outputs/GVL_COM.K4S2_02_E18_stComOut/D[10] <-> COM Outputs/Data Out 10
//     ComTask Outputs/GVL_COM.K4S2_02_E18_stComOut/D[11] <-> COM Outputs/Data Out 11
//     ComTask Outputs/GVL_COM.K4S2_02_E18_stComOut/D[12] <-> COM Outputs/Data Out 12
//     ComTask Outputs/GVL_COM.K4S2_02_E18_stComOut/D[13] <-> COM Outputs/Data Out 13
//     ComTask Outputs/GVL_COM.K4S2_02_E18_stComOut/D[14] <-> COM Outputs/Data Out 14
//     ComTask Outputs/GVL_COM.K4S2_02_E18_stComOut/D[15] <-> COM Outputs/Data Out 15
//     ComTask Outputs/GVL_COM.K4S2_02_E18_stComOut/D[16] <-> COM Outputs/Data Out 16
//     ComTask Outputs/GVL_COM.K4S2_02_E18_stComOut/D[17] <-> COM Outputs/Data Out 17
//     ComTask Outputs/GVL_COM.K4S2_02_E18_stComOut/D[18] <-> COM Outputs/Data Out 18
//     ComTask Outputs/GVL_COM.K4S2_02_E18_stComOut/D[19] <-> COM Outputs/Data Out 19
//     ComTask Outputs/GVL_COM.K4S2_02_E18_stComOut/D[1] <-> COM Outputs/Data Out 1
//     ComTask Outputs/GVL_COM.K4S2_02_E18_stComOut/D[20] <-> COM Outputs/Data Out 20
//     ComTask Outputs/GVL_COM.K4S2_02_E18_stComOut/D[21] <-> COM Outputs/Data Out 21
//     ComTask Outputs/GVL_COM.K4S2_02_E18_stComOut/D[2] <-> COM Outputs/Data Out 2
//     ComTask Outputs/GVL_COM.K4S2_02_E18_stComOut/D[3] <-> COM Outputs/Data Out 3
//     ComTask Outputs/GVL_COM.K4S2_02_E18_stComOut/D[4] <-> COM Outputs/Data Out 4
//     ComTask Outputs/GVL_COM.K4S2_02_E18_stComOut/D[5] <-> COM Outputs/Data Out 5
//     ComTask Outputs/GVL_COM.K4S2_02_E18_stComOut/D[6] <-> COM Outputs/Data Out 6
//     ComTask Outputs/GVL_COM.K4S2_02_E18_stComOut/D[7] <-> COM Outputs/Data Out 7
//     ComTask Outputs/GVL_COM.K4S2_02_E18_stComOut/D[8] <-> COM Outputs/Data Out 8
//     ComTask Outputs/GVL_COM.K4S2_02_E18_stComOut/D[9] <-> COM Outputs/Data Out 9
//   PLC_TMO_VAC Instance <-> Device 1 (EtherCAT)/TMO_K4S2_DRL_02 (EK1100)/K4S2_02_E19 (EL1004)
//     PlcTask Inputs/GVL_Hutch_Valves.TMO_ROUGH1_VRC_01.i_xClsLS <-> Channel 2/Input
//     PlcTask Inputs/GVL_Hutch_Valves.TMO_ROUGH2_VRC_01.i_xClsLS <-> Channel 4/Input
//     PlcTask Inputs/GVL_Hutch_Valves.TMO_ROUGH1_VRC_01.i_xOpnLS <-> Channel 1/Input
//     PlcTask Inputs/GVL_Hutch_Valves.TMO_ROUGH2_VRC_01.i_xOpnLS <-> Channel 3/Input
//   PLC_TMO_VAC Instance <-> Device 1 (EtherCAT)/TMO_K4S2_DRL_02 (EK1100)/K4S2_02_E2 (EL3174)
//     PlcTask Inputs/GVL_Hutch_Gauges.IM4K4_PPM_GCC_01.i_iPRESS_R <-> AI Standard Channel 2/Value
//     PlcTask Inputs/GVL_Hutch_Gauges.PA1K4_IP1_GPI_01.i_iPRESS_R <-> AI Standard Channel 1/Value
//   PLC_TMO_VAC Instance <-> Device 1 (EtherCAT)/TMO_K4S2_DRL_02 (EK1100)/K4S2_02_E20 (EL2004)
//     PlcTask Outputs/GVL_Hutch_Valves.TMO_ROUGH1_VRC_01.q_xOPN_DO <-> Channel 1/Output
//     PlcTask Outputs/GVL_Hutch_Valves.TMO_ROUGH2_VRC_01.q_xOPN_DO <-> Channel 2/Output
//   PLC_TMO_VAC Instance <-> Device 1 (EtherCAT)/TMO_K4S2_DRL_02 (EK1100)/K4S2_02_E5 (EL2624)
//     PlcTask Outputs/GVL_Hutch_Gauges.IM4K4_PPM_GCC_01.q_xHV_DIS <-> Channel 4/Output
//     PlcTask Outputs/GVL_Hutch_Gauges.MR2K4_KBO_GCC_01.q_xHV_DIS <-> Channel 2/Output
//     PlcTask Outputs/GVL_Hutch_Gauges.PA1K4_IP1_GCC_01.q_xHV_DIS <-> Channel 3/Output
//   PLC_TMO_VAC Instance <-> Device 1 (EtherCAT)/TMO_K4S2_DRL_02 (EK1100)/K4S2_02_E7 (EL1124)
//     PlcTask Inputs/GVL_Hutch_Gauges.MR2K4_KBO_GCC_01.i_xDisc_Active <-> Channel 4/Input
//     PlcTask Inputs/GVL_Hutch_Gauges.MR2K4_KBO_GCC_01.i_xHV_ON <-> Channel 3/Input
//   PLC_TMO_VAC Instance <-> Device 1 (EtherCAT)/TMO_K4S2_DRL_02 (EK1100)/K4S2_02_E8 (EL1124)
//     PlcTask Inputs/GVL_Hutch_Gauges.IM4K4_PPM_GCC_01.i_xDisc_Active <-> Channel 4/Input
//     PlcTask Inputs/GVL_Hutch_Gauges.IM4K4_PPM_GCC_01.i_xHV_ON <-> Channel 3/Input
//     PlcTask Inputs/GVL_Hutch_Gauges.PA1K4_IP1_GCC_01.i_xDisc_Active <-> Channel 2/Input
//     PlcTask Inputs/GVL_Hutch_Gauges.PA1K4_IP1_GCC_01.i_xHV_ON <-> Channel 1/Input
//   PLC_TMO_VAC Instance <-> Device 1 (EtherCAT)/TMO_K4S6_ EP1 (EP4374-0002)
//     PlcTask Inputs/GVL_Hutch_Gauges.TMO_ROUGH1_GPI_03.i_iPRESS_R <-> AI Inputs Channel 1/Value
//     PlcTask Outputs/GVL_Hutch_Valves.TMO_ROUGH1_VFV_03.q_iRawPosition <-> AO Outputs Channel 3/Analog output
//   PLC_TMO_VAC Instance <-> Device 1 (EtherCAT)/TMO_K4S6_DRL_01 (EK1100)/K4S6_01_E1 (EL1004)
//     PlcTask Inputs/GVL_Hutch_Valves.TMO_ROUGH1_VRC_02.i_xClsLS <-> Channel 2/Input
//     PlcTask Inputs/GVL_Hutch_Valves.TMO_ROUGH1_VRC_02.i_xOpnLS <-> Channel 1/Input
//   PLC_TMO_VAC Instance <-> Device 1 (EtherCAT)/TMO_K4S6_DRL_01 (EK1100)/K4S6_01_E11 (EL1004)
//     PlcTask Inputs/GVL_Hutch_Pumps.IM5K4_PPM_PTM_01.i_xFaultNC <-> Channel 1/Input
//   PLC_TMO_VAC Instance <-> Device 1 (EtherCAT)/TMO_K4S6_DRL_01 (EK1100)/K4S6_01_E12 (EL2004)
//     PlcTask Outputs/GVL_Hutch_Pumps.IM5K4_PPM_PTM_01.q_PumpingStation <-> Channel 1/Output
//   PLC_TMO_VAC Instance <-> Device 1 (EtherCAT)/TMO_K4S6_DRL_01 (EK1100)/K4S6_01_E14 (EL2624)
//     PlcTask Outputs/GVL_Hutch_Gauges.IM5K4_PPM_GCC_01.q_xHV_DIS <-> Channel 2/Output
//     PlcTask Outputs/GVL_Hutch_Gauges.MR4K4_KBO_GCC_01.q_xHV_DIS <-> Channel 4/Output
//     PlcTask Outputs/GVL_Hutch_Gauges.PA2K4_IP1_GCC_01.q_xHV_DIS <-> Channel 3/Output
//     PlcTask Outputs/GVL_Hutch_Gauges.TM1K4_GCC_01.q_xHV_DIS <-> Channel 1/Output
//   PLC_TMO_VAC Instance <-> Device 1 (EtherCAT)/TMO_K4S6_DRL_01 (EK1100)/K4S6_01_E15 (EL3174)
//     PlcTask Inputs/GVL_Hutch_Gauges.IM5K4_PPM_GCC_01.i_iPRESS_R <-> AI Standard Channel 2/Value
//     PlcTask Inputs/GVL_Hutch_Gauges.PA2K4_IP1_GCC_01.i_iPRESS_R <-> AI Standard Channel 3/Value
//     PlcTask Inputs/GVL_Hutch_Gauges.PA2K4_IP1_GPI_01.i_iPRESS_R <-> AI Standard Channel 4/Value
//     PlcTask Inputs/GVL_Hutch_Gauges.TM1K4_GCC_01.i_iPRESS_R <-> AI Standard Channel 1/Value
//   PLC_TMO_VAC Instance <-> Device 1 (EtherCAT)/TMO_K4S6_DRL_01 (EK1100)/K4S6_01_E18 (EL3174)
//     PlcTask Inputs/GVL_Hutch_Gauges.MR4K4_KBO_GCC_01.i_iPRESS_R <-> AI Standard Channel 2/Value
//     PlcTask Inputs/GVL_Hutch_Gauges.MR4K4_KBO_GPI_01.i_iPRESS_R <-> AI Standard Channel 1/Value
//   PLC_TMO_VAC Instance <-> Device 1 (EtherCAT)/TMO_K4S6_DRL_01 (EK1100)/K4S6_01_E2 (EL2004)
//     PlcTask Outputs/GVL_Hutch_Valves.TMO_ROUGH1_VRC_02.q_xOPN_DO <-> Channel 1/Output
//   PLC_TMO_VAC Instance <-> Device 1 (EtherCAT)/TMO_K4S6_DRL_01 (EK1100)/K4S6_01_E20 (EL1124)
//     PlcTask Inputs/GVL_Hutch_Gauges.IM5K4_PPM_GCC_01.i_xDisc_Active <-> Channel 4/Input
//     PlcTask Inputs/GVL_Hutch_Gauges.IM5K4_PPM_GCC_01.i_xHV_ON <-> Channel 3/Input
//     PlcTask Inputs/GVL_Hutch_Gauges.TM1K4_GCC_01.i_xDisc_Active <-> Channel 2/Input
//     PlcTask Inputs/GVL_Hutch_Gauges.TM1K4_GCC_01.i_xHV_ON <-> Channel 1/Input
//   PLC_TMO_VAC Instance <-> Device 1 (EtherCAT)/TMO_K4S6_DRL_01 (EK1100)/K4S6_01_E21 (EL1124)
//     PlcTask Inputs/GVL_Hutch_Gauges.MR4K4_KBO_GCC_01.i_xDisc_Active <-> Channel 4/Input
//     PlcTask Inputs/GVL_Hutch_Gauges.MR4K4_KBO_GCC_01.i_xHV_ON <-> Channel 3/Input
//     PlcTask Inputs/GVL_Hutch_Gauges.PA2K4_IP1_GCC_01.i_xDisc_Active <-> Channel 2/Input
//     PlcTask Inputs/GVL_Hutch_Gauges.PA2K4_IP1_GCC_01.i_xHV_ON <-> Channel 1/Input
//   PLC_TMO_VAC Instance <-> Device 1 (EtherCAT)/TMO_K4S6_DRL_01 (EK1100)/K4S6_01_E22_IP1 (EL1004)
//     PlcTask Inputs/GVL_Variables.xLAMP_PTM_NOK <-> Channel 1/Input
//   PLC_TMO_VAC Instance <-> Device 1 (EtherCAT)/TMO_K4S6_DRL_01 (EK1100)/K4S6_01_E3 (EL1004)
//     PlcTask Inputs/GVL_Hutch_Valves.LI3K4_IP1_VWC_01.i_xClsLS <-> Channel 2/Input
//     PlcTask Inputs/GVL_Hutch_Valves.LI3K4_IP1_VWC_01.i_xOpnLS <-> Channel 1/Input
//     PlcTask Inputs/GVL_Hutch_Valves.PC5K4_VWC_01.i_xClsLS <-> Channel 4/Input
//     PlcTask Inputs/GVL_Hutch_Valves.PC5K4_VWC_01.i_xOpnLS <-> Channel 3/Input
//   PLC_TMO_VAC Instance <-> Device 1 (EtherCAT)/TMO_K4S6_DRL_01 (EK1100)/K4S6_01_E4 (EL2004)
//     PlcTask Outputs/GVL_Hutch_Valves.LI3K4_IP1_VWC_01.q_xOPN_DO <-> Channel 1/Output
//     PlcTask Outputs/GVL_Hutch_Valves.PC5K4_VWC_01.q_xOPN_DO <-> Channel 2/Output
//   PLC_TMO_VAC Instance <-> Device 1 (EtherCAT)/TMO_K4S6_DRL_01 (EK1100)/K4S6_01_E5 (EL6021)
//     ComTask Inputs/GVL_COM.K4S6_01_E5_stComIn/D[0] <-> COM TxPDO-Map Inputs/Data In 0
//     ComTask Inputs/GVL_COM.K4S6_01_E5_stComIn/D[10] <-> COM TxPDO-Map Inputs/Data In 10
//     ComTask Inputs/GVL_COM.K4S6_01_E5_stComIn/D[11] <-> COM TxPDO-Map Inputs/Data In 11
//     ComTask Inputs/GVL_COM.K4S6_01_E5_stComIn/D[12] <-> COM TxPDO-Map Inputs/Data In 12
//     ComTask Inputs/GVL_COM.K4S6_01_E5_stComIn/D[13] <-> COM TxPDO-Map Inputs/Data In 13
//     ComTask Inputs/GVL_COM.K4S6_01_E5_stComIn/D[14] <-> COM TxPDO-Map Inputs/Data In 14
//     ComTask Inputs/GVL_COM.K4S6_01_E5_stComIn/D[15] <-> COM TxPDO-Map Inputs/Data In 15
//     ComTask Inputs/GVL_COM.K4S6_01_E5_stComIn/D[16] <-> COM TxPDO-Map Inputs/Data In 16
//     ComTask Inputs/GVL_COM.K4S6_01_E5_stComIn/D[17] <-> COM TxPDO-Map Inputs/Data In 17
//     ComTask Inputs/GVL_COM.K4S6_01_E5_stComIn/D[18] <-> COM TxPDO-Map Inputs/Data In 18
//     ComTask Inputs/GVL_COM.K4S6_01_E5_stComIn/D[19] <-> COM TxPDO-Map Inputs/Data In 19
//     ComTask Inputs/GVL_COM.K4S6_01_E5_stComIn/D[1] <-> COM TxPDO-Map Inputs/Data In 1
//     ComTask Inputs/GVL_COM.K4S6_01_E5_stComIn/D[20] <-> COM TxPDO-Map Inputs/Data In 20
//     ComTask Inputs/GVL_COM.K4S6_01_E5_stComIn/D[21] <-> COM TxPDO-Map Inputs/Data In 21
//     ComTask Inputs/GVL_COM.K4S6_01_E5_stComIn/D[2] <-> COM TxPDO-Map Inputs/Data In 2
//     ComTask Inputs/GVL_COM.K4S6_01_E5_stComIn/D[3] <-> COM TxPDO-Map Inputs/Data In 3
//     ComTask Inputs/GVL_COM.K4S6_01_E5_stComIn/D[4] <-> COM TxPDO-Map Inputs/Data In 4
//     ComTask Inputs/GVL_COM.K4S6_01_E5_stComIn/D[5] <-> COM TxPDO-Map Inputs/Data In 5
//     ComTask Inputs/GVL_COM.K4S6_01_E5_stComIn/D[6] <-> COM TxPDO-Map Inputs/Data In 6
//     ComTask Inputs/GVL_COM.K4S6_01_E5_stComIn/D[7] <-> COM TxPDO-Map Inputs/Data In 7
//     ComTask Inputs/GVL_COM.K4S6_01_E5_stComIn/D[8] <-> COM TxPDO-Map Inputs/Data In 8
//     ComTask Inputs/GVL_COM.K4S6_01_E5_stComIn/D[9] <-> COM TxPDO-Map Inputs/Data In 9
//     ComTask Inputs/GVL_COM.K4S6_01_E5_stComIn/Status <-> COM TxPDO-Map Inputs/Status
//     ComTask Outputs/GVL_COM.K4S6_01_E5_stComOut/Ctrl <-> COM RxPDO-Map Outputs/Ctrl
//     ComTask Outputs/GVL_COM.K4S6_01_E5_stComOut/D[0] <-> COM RxPDO-Map Outputs/Data Out 0
//     ComTask Outputs/GVL_COM.K4S6_01_E5_stComOut/D[10] <-> COM RxPDO-Map Outputs/Data Out 10
//     ComTask Outputs/GVL_COM.K4S6_01_E5_stComOut/D[11] <-> COM RxPDO-Map Outputs/Data Out 11
//     ComTask Outputs/GVL_COM.K4S6_01_E5_stComOut/D[12] <-> COM RxPDO-Map Outputs/Data Out 12
//     ComTask Outputs/GVL_COM.K4S6_01_E5_stComOut/D[13] <-> COM RxPDO-Map Outputs/Data Out 13
//     ComTask Outputs/GVL_COM.K4S6_01_E5_stComOut/D[14] <-> COM RxPDO-Map Outputs/Data Out 14
//     ComTask Outputs/GVL_COM.K4S6_01_E5_stComOut/D[15] <-> COM RxPDO-Map Outputs/Data Out 15
//     ComTask Outputs/GVL_COM.K4S6_01_E5_stComOut/D[16] <-> COM RxPDO-Map Outputs/Data Out 16
//     ComTask Outputs/GVL_COM.K4S6_01_E5_stComOut/D[17] <-> COM RxPDO-Map Outputs/Data Out 17
//     ComTask Outputs/GVL_COM.K4S6_01_E5_stComOut/D[18] <-> COM RxPDO-Map Outputs/Data Out 18
//     ComTask Outputs/GVL_COM.K4S6_01_E5_stComOut/D[19] <-> COM RxPDO-Map Outputs/Data Out 19
//     ComTask Outputs/GVL_COM.K4S6_01_E5_stComOut/D[1] <-> COM RxPDO-Map Outputs/Data Out 1
//     ComTask Outputs/GVL_COM.K4S6_01_E5_stComOut/D[20] <-> COM RxPDO-Map Outputs/Data Out 20
//     ComTask Outputs/GVL_COM.K4S6_01_E5_stComOut/D[21] <-> COM RxPDO-Map Outputs/Data Out 21
//     ComTask Outputs/GVL_COM.K4S6_01_E5_stComOut/D[2] <-> COM RxPDO-Map Outputs/Data Out 2
//     ComTask Outputs/GVL_COM.K4S6_01_E5_stComOut/D[3] <-> COM RxPDO-Map Outputs/Data Out 3
//     ComTask Outputs/GVL_COM.K4S6_01_E5_stComOut/D[4] <-> COM RxPDO-Map Outputs/Data Out 4
//     ComTask Outputs/GVL_COM.K4S6_01_E5_stComOut/D[5] <-> COM RxPDO-Map Outputs/Data Out 5
//     ComTask Outputs/GVL_COM.K4S6_01_E5_stComOut/D[6] <-> COM RxPDO-Map Outputs/Data Out 6
//     ComTask Outputs/GVL_COM.K4S6_01_E5_stComOut/D[7] <-> COM RxPDO-Map Outputs/Data Out 7
//     ComTask Outputs/GVL_COM.K4S6_01_E5_stComOut/D[8] <-> COM RxPDO-Map Outputs/Data Out 8
//     ComTask Outputs/GVL_COM.K4S6_01_E5_stComOut/D[9] <-> COM RxPDO-Map Outputs/Data Out 9
//   PLC_TMO_VAC Instance <-> Device 1 (EtherCAT)/TMO_K4S6_DRL_01 (EK1100)/K4S6_01_E6 (EL1004)
//     PlcTask Inputs/GVL_Hutch_Pumps.LI3K4_IP1_OUT_PTM_01.i_xAtSpd <-> Channel 1/Input
//     PlcTask Inputs/GVL_Hutch_Pumps.LI3K4_IP1_OUT_PTM_01.i_xFaultNC <-> Channel 3/Input
//     PlcTask Inputs/GVL_Hutch_Pumps.LI3K4_IP1_OUT_PTM_01.i_xRemote <-> Channel 2/Input
//     PlcTask Inputs/GVL_Hutch_Pumps.TM1K4_PTM_01.i_xAtSpd <-> Channel 4/Input
//   PLC_TMO_VAC Instance <-> Device 1 (EtherCAT)/TMO_K4S6_DRL_01 (EK1100)/K4S6_01_E7 (EL2004)
//     PlcTask Outputs/GVL_Hutch_Pumps.LI3K4_IP1_OUT_PTM_01.q_PumpingStation <-> Channel 3/Output
//     PlcTask Outputs/GVL_Hutch_Pumps.LI3K4_IP1_OUT_PTM_01.q_RunDO <-> Channel 1/Output
//     PlcTask Outputs/GVL_Hutch_Pumps.LI3K4_IP1_OUT_PTM_01.q_xRemote <-> Channel 2/Output
//     PlcTask Outputs/GVL_Hutch_Pumps.TM1K4_PTM_01.q_RunDO <-> Channel 4/Output
//   PLC_TMO_VAC Instance <-> Device 1 (EtherCAT)/TMO_K4S6_DRL_01 (EK1100)/K4S6_01_E8 (EL1004)
//     PlcTask Inputs/GVL_Hutch_Pumps.IM5K4_PPM_PTM_01.i_xAtSpd <-> Channel 3/Input
//     PlcTask Inputs/GVL_Hutch_Pumps.IM5K4_PPM_PTM_01.i_xRemote <-> Channel 4/Input
//     PlcTask Inputs/GVL_Hutch_Pumps.TM1K4_PTM_01.i_xFaultNC <-> Channel 2/Input
//     PlcTask Inputs/GVL_Hutch_Pumps.TM1K4_PTM_01.i_xRemote <-> Channel 1/Input
//   PLC_TMO_VAC Instance <-> Device 1 (EtherCAT)/TMO_K4S6_DRL_01 (EK1100)/K4S6_01_E9 (EL2004)
//     PlcTask Outputs/GVL_Hutch_Pumps.IM5K4_PPM_PTM_01.q_RunDO <-> Channel 3/Output
//     PlcTask Outputs/GVL_Hutch_Pumps.IM5K4_PPM_PTM_01.q_xRemote <-> Channel 4/Output
//     PlcTask Outputs/GVL_Hutch_Pumps.TM1K4_PTM_01.q_PumpingStation <-> Channel 2/Output
//     PlcTask Outputs/GVL_Hutch_Pumps.TM1K4_PTM_01.q_xRemote <-> Channel 1/Output
//   PLC_TMO_VAC Instance <-> Device 1 (EtherCAT)/TMO_K4S8_DRL_01 (EK1100)/K4S8_01_E1 (EL1004)
//     FSVTask Inputs/GVL_FS_Devices.MR4K4_KBO_VFS_1.i_xClsLS <-> Channel 1/Input
//     FSVTask Inputs/GVL_FS_Devices.MR4K4_KBO_VFS_1.i_xOpnLS <-> Channel 2/Input
//   PLC_TMO_VAC Instance <-> Device 1 (EtherCAT)/TMO_K4S8_DRL_01 (EK1100)/K4S8_01_E3 (EL2202)
//     FSVTask Outputs/GVL_FS_Devices.MR4K4_KBO_VFS_1.q_xClose_A <-> Channel 1/Output
//     FSVTask Outputs/GVL_FS_Devices.MR4K4_KBO_VFS_1.q_xClose_B <-> Channel 2/Output
//   PLC_TMO_VAC Instance <-> Device 1 (EtherCAT)/TMO_K4S8_DRL_01 (EK1100)/K4S8_01_E4 (EL2202)
//     FSVTask Outputs/GVL_FS_Devices.MR4K4_KBO_VFS_1.q_xClose_C <-> Channel 1/Output
//     FSVTask Outputs/GVL_FS_Devices.MR4K4_KBO_VFS_1.q_xOPN_DO <-> Channel 2/Output
//   PLC_TMO_VAC Instance <-> Device 1 (EtherCAT)/TMO_K4S8_DRL_01 (EK1100)/K4S8_01_E5 (EL1004)
//     PlcTask Inputs/GVL_Hutch_Valves.MR4K4_KBO_VWC_01.i_xClsLS <-> Channel 2/Input
//     PlcTask Inputs/GVL_Hutch_Valves.MR5K4_KBO_VWC_01.i_xClsLS <-> Channel 4/Input
//     PlcTask Inputs/GVL_Hutch_Valves.MR4K4_KBO_VWC_01.i_xOpnLS <-> Channel 1/Input
//     PlcTask Inputs/GVL_Hutch_Valves.MR5K4_KBO_VWC_01.i_xOpnLS <-> Channel 3/Input
//   PLC_TMO_VAC Instance <-> Device 1 (EtherCAT)/TMO_K4S8_DRL_01 (EK1100)/K4S8_01_E6 (EL2004)
//     PlcTask Outputs/GVL_Hutch_Valves.MR4K4_KBO_VWC_01.q_xOPN_DO <-> Channel 1/Output
//     PlcTask Outputs/GVL_Hutch_Valves.MR5K4_KBO_VWC_01.q_xOPN_DO <-> Channel 2/Output
//   PLC_TMO_VAC Instance <-> Device 1 (EtherCAT)/TMO_WALL_WEST_EP01 (EP4374-0002)
//     PlcTask Inputs/GVL_Hutch_Gauges.TMO_ROUGH1_GPI_01.i_iPRESS_R <-> AI Inputs Channel 1/Value
//     PlcTask Inputs/GVL_Hutch_Gauges.TMO_ROUGH2_GPI_01.i_iPRESS_R <-> AI Inputs Channel 2/Value
//     PlcTask Outputs/GVL_Hutch_Valves.TMO_ROUGH1_VFV_01.q_iRawPosition <-> AO Outputs Channel 3/Analog output
//   PLC_TMO_VAC Instance <-> PLC_TMO_VAC/PLC_TMO_VAC Instance
//     FSVTask Inputs/GVL_FS_Devices.MR3K4_KBO_VFS_1.i_xCLS_SW <-> PlcTask Outputs/GVL_FS_Devices.MR3K4_KBO_VFS_Interface.q_xCLS_SW
//     FSVTask Inputs/GVL_FS_Devices.MR4K4_KBO_VFS_1.i_xCLS_SW <-> PlcTask Outputs/GVL_FS_Devices.MR4K4_KBO_VFS_Interface.q_xCLS_SW
//     FSVTask Inputs/GVL_FS_Devices.MR3K4_KBO_VFS_1.i_xOPN_SW <-> PlcTask Outputs/GVL_FS_Devices.MR3K4_KBO_VFS_Interface.q_xOPN_SW
//     FSVTask Inputs/GVL_FS_Devices.MR4K4_KBO_VFS_1.i_xOPN_SW <-> PlcTask Outputs/GVL_FS_Devices.MR4K4_KBO_VFS_Interface.q_xOPN_SW
//     FSVTask Inputs/GVL_FS_Devices.MR3K4_KBO_VFS_1.i_xOverrideMode <-> PlcTask Outputs/GVL_FS_Devices.MR3K4_KBO_VFS_Interface.q_xOverrideMode
//     FSVTask Inputs/GVL_FS_Devices.MR4K4_KBO_VFS_1.i_xOverrideMode <-> PlcTask Outputs/GVL_FS_Devices.MR4K4_KBO_VFS_Interface.q_xOverrideMode
//     FSVTask Inputs/GVL_FS_Devices.MR3K4_KBO_VFS_1.i_xOverrideOpen <-> PlcTask Outputs/GVL_FS_Devices.MR3K4_KBO_VFS_Interface.q_xOverrideOpen
//     FSVTask Inputs/GVL_FS_Devices.MR4K4_KBO_VFS_1.i_xOverrideOpen <-> PlcTask Outputs/GVL_FS_Devices.MR4K4_KBO_VFS_Interface.q_xOverrideOpen
//     FSVTask Inputs/GVL_FS_Devices.MR3K4_KBO_VFS_1.i_xPress_OK <-> PlcTask Outputs/GVL_FS_Devices.MR3K4_KBO_VFS_Interface.q_xPRESS_OK
//     FSVTask Inputs/GVL_FS_Devices.MR4K4_KBO_VFS_1.i_xPress_OK <-> PlcTask Outputs/GVL_FS_Devices.MR4K4_KBO_VFS_Interface.q_xPRESS_OK
//     FSVTask Inputs/GVL_FS_Devices.MR3K4_KBO_VFS_1.i_xVAC_FAULT_Reset <-> PlcTask Outputs/GVL_FS_Devices.MR3K4_KBO_VFS_Interface.q_xVAC_FAULT_Reset
//     FSVTask Inputs/GVL_FS_Devices.MR4K4_KBO_VFS_1.i_xVAC_FAULT_Reset <-> PlcTask Outputs/GVL_FS_Devices.MR4K4_KBO_VFS_Interface.q_xVAC_FAULT_Reset
//     FSVTask Inputs/GVL_FS_Devices.TV1K4_VFS_1.i_xCLS_SW <-> PlcTask Outputs/GVL_FS_Devices.TV1K4_VFS_Interface.q_xCLS_SW
//     FSVTask Inputs/GVL_FS_Devices.TV1K4_VFS_1.i_xOPN_SW <-> PlcTask Outputs/GVL_FS_Devices.TV1K4_VFS_Interface.q_xOPN_SW
//     FSVTask Inputs/GVL_FS_Devices.TV1K4_VFS_1.i_xOverrideMode <-> PlcTask Outputs/GVL_FS_Devices.TV1K4_VFS_Interface.q_xOverrideMode
//     FSVTask Inputs/GVL_FS_Devices.TV1K4_VFS_1.i_xOverrideOpen <-> PlcTask Outputs/GVL_FS_Devices.TV1K4_VFS_Interface.q_xOverrideOpen
//     FSVTask Inputs/GVL_FS_Devices.TV1K4_VFS_1.i_xPress_OK <-> PlcTask Outputs/GVL_FS_Devices.TV1K4_VFS_Interface.q_xPRESS_OK
//     FSVTask Inputs/GVL_FS_Devices.TV1K4_VFS_1.i_xVAC_FAULT_Reset <-> PlcTask Outputs/GVL_FS_Devices.TV1K4_VFS_Interface.q_xVAC_FAULT_Reset
//     FSVTask Outputs/GVL_FS_Devices.MR3K4_KBO_VFS_1.q_eVFS_State <-> PlcTask Inputs/GVL_FS_Devices.MR3K4_KBO_VFS_Interface.i_eVFS_State
//     FSVTask Outputs/GVL_FS_Devices.MR4K4_KBO_VFS_1.q_eVFS_State <-> PlcTask Inputs/GVL_FS_Devices.MR4K4_KBO_VFS_Interface.i_eVFS_State
//     FSVTask Outputs/GVL_FS_Devices.MR3K4_KBO_VFS_1.q_xMPS_OK <-> PlcTask Inputs/GVL_FS_Devices.MR3K4_KBO_VFS_Interface.i_xMPS_OK
//     FSVTask Outputs/GVL_FS_Devices.MR4K4_KBO_VFS_1.q_xMPS_OK <-> PlcTask Inputs/GVL_FS_Devices.MR4K4_KBO_VFS_Interface.i_xMPS_OK
//     FSVTask Outputs/GVL_FS_Devices.MR3K4_KBO_VFS_1.q_xVAC_FAULT_OK <-> PlcTask Inputs/GVL_FS_Devices.MR3K4_KBO_VFS_Interface.i_xVAC_FAULT_OK
//     FSVTask Outputs/GVL_FS_Devices.MR4K4_KBO_VFS_1.q_xVAC_FAULT_OK <-> PlcTask Inputs/GVL_FS_Devices.MR4K4_KBO_VFS_Interface.i_xVAC_FAULT_OK
//     FSVTask Outputs/GVL_FS_Devices.MR3K4_KBO_VFS_1.q_xVFS_Closed <-> PlcTask Inputs/GVL_FS_Devices.MR3K4_KBO_VFS_Interface.i_xVFS_Closed
//     FSVTask Outputs/GVL_FS_Devices.MR4K4_KBO_VFS_1.q_xVFS_Closed <-> PlcTask Inputs/GVL_FS_Devices.MR4K4_KBO_VFS_Interface.i_xVFS_Closed
//     FSVTask Outputs/GVL_FS_Devices.TV1K4_VFS_1.q_eVFS_State <-> PlcTask Inputs/GVL_FS_Devices.TV1K4_VFS_Interface.i_eVFS_State
//     FSVTask Outputs/GVL_FS_Devices.TV1K4_VFS_1.q_xMPS_OK <-> PlcTask Inputs/GVL_FS_Devices.TV1K4_VFS_Interface.i_xMPS_OK
//     FSVTask Outputs/GVL_FS_Devices.TV1K4_VFS_1.q_xVAC_FAULT_OK <-> PlcTask Inputs/GVL_FS_Devices.TV1K4_VFS_Interface.i_xVAC_FAULT_OK
//     FSVTask Outputs/GVL_FS_Devices.TV1K4_VFS_1.q_xVFS_Closed <-> PlcTask Inputs/GVL_FS_Devices.TV1K4_VFS_Interface.i_xVFS_Closed
//     PlcTask Inputs/GVL_FS_Devices.MR3K4_KBO_VFS_Interface.i_eVFS_State <-> FSVTask Outputs/GVL_FS_Devices.MR3K4_KBO_VFS_1.q_eVFS_State
//     PlcTask Inputs/GVL_FS_Devices.MR4K4_KBO_VFS_Interface.i_eVFS_State <-> FSVTask Outputs/GVL_FS_Devices.MR4K4_KBO_VFS_1.q_eVFS_State
//     PlcTask Inputs/GVL_FS_Devices.MR3K4_KBO_VFS_Interface.i_xMPS_OK <-> FSVTask Outputs/GVL_FS_Devices.MR3K4_KBO_VFS_1.q_xMPS_OK
//     PlcTask Inputs/GVL_FS_Devices.MR4K4_KBO_VFS_Interface.i_xMPS_OK <-> FSVTask Outputs/GVL_FS_Devices.MR4K4_KBO_VFS_1.q_xMPS_OK
//     PlcTask Inputs/GVL_FS_Devices.MR3K4_KBO_VFS_Interface.i_xVAC_FAULT_OK <-> FSVTask Outputs/GVL_FS_Devices.MR3K4_KBO_VFS_1.q_xVAC_FAULT_OK
//     PlcTask Inputs/GVL_FS_Devices.MR4K4_KBO_VFS_Interface.i_xVAC_FAULT_OK <-> FSVTask Outputs/GVL_FS_Devices.MR4K4_KBO_VFS_1.q_xVAC_FAULT_OK
//     PlcTask Inputs/GVL_FS_Devices.MR3K4_KBO_VFS_Interface.i_xVFS_Closed <-> FSVTask Outputs/GVL_FS_Devices.MR3K4_KBO_VFS_1.q_xVFS_Closed
//     PlcTask Inputs/GVL_FS_Devices.MR4K4_KBO_VFS_Interface.i_xVFS_Closed <-> FSVTask Outputs/GVL_FS_Devices.MR4K4_KBO_VFS_1.q_xVFS_Closed
//     PlcTask Inputs/GVL_FS_Devices.TV1K4_VFS_Interface.i_eVFS_State <-> FSVTask Outputs/GVL_FS_Devices.TV1K4_VFS_1.q_eVFS_State
//     PlcTask Inputs/GVL_FS_Devices.TV1K4_VFS_Interface.i_xMPS_OK <-> FSVTask Outputs/GVL_FS_Devices.TV1K4_VFS_1.q_xMPS_OK
//     PlcTask Inputs/GVL_FS_Devices.TV1K4_VFS_Interface.i_xVAC_FAULT_OK <-> FSVTask Outputs/GVL_FS_Devices.TV1K4_VFS_1.q_xVAC_FAULT_OK
//     PlcTask Inputs/GVL_FS_Devices.TV1K4_VFS_Interface.i_xVFS_Closed <-> FSVTask Outputs/GVL_FS_Devices.TV1K4_VFS_1.q_xVFS_Closed
//     PlcTask Outputs/GVL_FS_Devices.MR3K4_KBO_VFS_Interface.q_xCLS_SW <-> FSVTask Inputs/GVL_FS_Devices.MR3K4_KBO_VFS_1.i_xCLS_SW
//     PlcTask Outputs/GVL_FS_Devices.MR4K4_KBO_VFS_Interface.q_xCLS_SW <-> FSVTask Inputs/GVL_FS_Devices.MR4K4_KBO_VFS_1.i_xCLS_SW
//     PlcTask Outputs/GVL_FS_Devices.MR3K4_KBO_VFS_Interface.q_xOPN_SW <-> FSVTask Inputs/GVL_FS_Devices.MR3K4_KBO_VFS_1.i_xOPN_SW
//     PlcTask Outputs/GVL_FS_Devices.MR4K4_KBO_VFS_Interface.q_xOPN_SW <-> FSVTask Inputs/GVL_FS_Devices.MR4K4_KBO_VFS_1.i_xOPN_SW
//     PlcTask Outputs/GVL_FS_Devices.MR3K4_KBO_VFS_Interface.q_xOverrideMode <-> FSVTask Inputs/GVL_FS_Devices.MR3K4_KBO_VFS_1.i_xOverrideMode
//     PlcTask Outputs/GVL_FS_Devices.MR4K4_KBO_VFS_Interface.q_xOverrideMode <-> FSVTask Inputs/GVL_FS_Devices.MR4K4_KBO_VFS_1.i_xOverrideMode
//     PlcTask Outputs/GVL_FS_Devices.MR3K4_KBO_VFS_Interface.q_xOverrideOpen <-> FSVTask Inputs/GVL_FS_Devices.MR3K4_KBO_VFS_1.i_xOverrideOpen
//     PlcTask Outputs/GVL_FS_Devices.MR4K4_KBO_VFS_Interface.q_xOverrideOpen <-> FSVTask Inputs/GVL_FS_Devices.MR4K4_KBO_VFS_1.i_xOverrideOpen
//     PlcTask Outputs/GVL_FS_Devices.MR3K4_KBO_VFS_Interface.q_xPRESS_OK <-> FSVTask Inputs/GVL_FS_Devices.MR3K4_KBO_VFS_1.i_xPress_OK
//     PlcTask Outputs/GVL_FS_Devices.MR4K4_KBO_VFS_Interface.q_xPRESS_OK <-> FSVTask Inputs/GVL_FS_Devices.MR4K4_KBO_VFS_1.i_xPress_OK
//     PlcTask Outputs/GVL_FS_Devices.MR3K4_KBO_VFS_Interface.q_xVAC_FAULT_Reset <-> FSVTask Inputs/GVL_FS_Devices.MR3K4_KBO_VFS_1.i_xVAC_FAULT_Reset
//     PlcTask Outputs/GVL_FS_Devices.MR4K4_KBO_VFS_Interface.q_xVAC_FAULT_Reset <-> FSVTask Inputs/GVL_FS_Devices.MR4K4_KBO_VFS_1.i_xVAC_FAULT_Reset
//     PlcTask Outputs/GVL_FS_Devices.TV1K4_VFS_Interface.q_xCLS_SW <-> FSVTask Inputs/GVL_FS_Devices.TV1K4_VFS_1.i_xCLS_SW
//     PlcTask Outputs/GVL_FS_Devices.TV1K4_VFS_Interface.q_xOPN_SW <-> FSVTask Inputs/GVL_FS_Devices.TV1K4_VFS_1.i_xOPN_SW
//     PlcTask Outputs/GVL_FS_Devices.TV1K4_VFS_Interface.q_xOverrideMode <-> FSVTask Inputs/GVL_FS_Devices.TV1K4_VFS_1.i_xOverrideMode
//     PlcTask Outputs/GVL_FS_Devices.TV1K4_VFS_Interface.q_xOverrideOpen <-> FSVTask Inputs/GVL_FS_Devices.TV1K4_VFS_1.i_xOverrideOpen
//     PlcTask Outputs/GVL_FS_Devices.TV1K4_VFS_Interface.q_xPRESS_OK <-> FSVTask Inputs/GVL_FS_Devices.TV1K4_VFS_1.i_xPress_OK
//     PlcTask Outputs/GVL_FS_Devices.TV1K4_VFS_Interface.q_xVAC_FAULT_Reset <-> FSVTask Inputs/GVL_FS_Devices.TV1K4_VFS_1.i_xVAC_FAULT_Reset
//   PLC_TMO_VAC_FS Instance <-> Device 1 (EtherCAT)/B940_K4S20_EK0  (EK1100)/K4S20-E1-FSV (EL1004)
//     PlcTask Inputs/GVL_FS.TV1K4_VFS_01.i_xClsLS <-> Channel 1/Input
//     PlcTask Inputs/GVL_FS.TV1K4_VFS_01.i_xOpnLS <-> Channel 2/Input
//   PLC_TMO_VAC_FS Instance <-> Device 1 (EtherCAT)/B940_K4S20_EK0  (EK1100)/K4S20-E2-FSV (EL2202)
//     PlcTask Outputs/GVL_FS.TV1K4_VFS_01.q_xClose_A <-> Channel 1/Output
//     PlcTask Outputs/GVL_FS.TV1K4_VFS_01.q_xClose_B <-> Channel 2/Output
//   PLC_TMO_VAC_FS Instance <-> Device 1 (EtherCAT)/B940_K4S20_EK0  (EK1100)/K4S20-E3-FSV (EL2202)
//     PlcTask Outputs/GVL_FS.TV1K4_VFS_01.q_xClose_C <-> Channel 1/Output
//     PlcTask Outputs/GVL_FS.TV1K4_VFS_01.q_xOPN_DO <-> Channel 2/Output
//   PLC_TMO_VAC_FS Instance <-> Device 1 (EtherCAT)/B940_R20_EK0 (EK1100)/R20_EK0_E5 (EL1124)
//     PlcTask Inputs/GVL_FS.TV1K4_VFS_01.i_xTrigger <-> Channel 1/Input

// ---- GVLs/GVL_FEE_Device.TcGVL
//{attribute 'qualified_only'}
VAR_GLOBAL

(* upstream vacuum ok *)
   {attribute 'pytmc' :=' pv : USVAC:OK:HI '}
   {attribute 'TcLinkTo' := 	' := 	TIIB[CX0_E2_EXILK (EL1008)]^Channel 1^Input	'}	
   USVacOk_HI AT%I* : BOOL; (* upstream vacuum <10E-6, for mirror VGC interlock *)
 
 	{attribute 'pytmc' :=' pv : USVAC:OK:LO '}
   {attribute 'TcLinkTo' := 	'	:= 	TIIB[CX0_E2_EXILK (EL1008)]^Channel 3^Input	'}	  
   USVacOk_LO AT%I* : BOOL; (* upstream vacuum <10E-4, for Ion pump interlock *)


(* Isolation gate valves*)

	{attribute 'pytmc' :=' pv : TV1K4:VGC:01 '}
	{attribute 'TcLinkTo' := 	'.i_xOpnLS	:=	TIIB[B940_K4S20_EB1  (EP2338-0002)]^Channel 1^Input;
								 .i_xClsLS	:=	TIIB[B940_K4S20_EB1  (EP2338-0002)]^Channel 2^Input;
								.q_xOPN_DO	:=	TIIB[B940_K4S20_EB1  (EP2338-0002)]^Channel 11^Output'}
	TV1K4_VGC_01: FB_VGC;
	
	{attribute 'pytmc' :=' pv : TV1K4:VGC:02 '}
	{attribute 'TcLinkTo' := 	'.i_xOpnLS	:=	TIIB[B940_K4S20_EB1  (EP2338-0002)]^Channel 5^Input;
								 .i_xClsLS	:=	TIIB[B940_K4S20_EB1  (EP2338-0002)]^Channel 6^Input;
								 .q_xOPN_DO	:=	TIIB[B940_K4S20_EB1  (EP2338-0002)]^Channel 15^Output'}	
 	TV1K4_VGC_02: FB_VGC;

	{attribute 'pytmc' :=' pv : ST3K4:PPS:VGC:01 '}
	{attribute 'TcLinkTo' := 	'.i_xOpnLS	:=	TIIB[B940_K4S33_EB1 (EP2338-0002)]^Channel 1^Input;
								 .i_xClsLS	:=	TIIB[B940_K4S33_EB1 (EP2338-0002)]^Channel 2^Input;
								 .q_xOPN_DO	:=	TIIB[B940_K4S33_EB1 (EP2338-0002)]^Channel 11^Output'}	
	ST3K4_PPS_VGC_01 : FB_VGC;
	
(* Pirani & Cold Cathode*)

	

	{attribute 'pytmc' :=' pv : TV1K4:GPI:01 '}
	{attribute 'TcLinkTo' := 	'.i_iPRESS_R	:=	TIIB[B940_K4S20_EB2  (EP3174-0002)]^AI Standard Channel 1^Value	'}
	TV1K4_GPI_01 : FB_MKS275;
	
	
	{attribute 'pytmc' :=' pv : TV1K4:GCC:01 '}
	{attribute 'TcLinkTo' := 	'.i_iPRESS_R	:=	TIIB[B940_K4S20_EB2  (EP3174-0002)]^AI Standard Channel 2^Value;
								 .q_xHV_DIS		:= 	TIIB[B940_K4S20_EB3 (EP2624-0002)]^Channel 1^Output	'}	
	TV1K4_GCC_01 : FB_MKS500_EP;
	
	{attribute 'pytmc' :=' pv : ST1K4:TEST:GPI:01 '}
	{attribute 'TcLinkTo' := 	'.i_iPRESS_R	:=	TIIB[B940_K4S24_EB1 (EP3174-0002)]^AI Standard Channel 1^Value		'}
	ST1K4_TEST_GPI_01 : FB_MKS275;
	
			
	{attribute 'pytmc' :=' pv : ST1K4:TEST:GCC:01 '}
	{attribute 'TcLinkTo' := 	'.i_iPRESS_R	:=	TIIB[B940_K4S24_EB1 (EP3174-0002)]^AI Standard Channel 2^Value;
								 .q_xHV_DIS		:= 	TIIB[B940_K4S24_EB2 (EP2624-0002)]^Channel 1^Output	'}	
	ST1K4_TEST_GCC_01 : FB_MKS500_EP;
	
	
	{attribute 'pytmc' :=' pv : ST2K4:BCS:GPI:01 '}
	{attribute 'TcLinkTo' := 	'.i_iPRESS_R	:=	TIIB[B940_K4S28_EB1 (EP3174-0002)]^AI Standard Channel 1^Value	'}
	ST2K4_BCS_GPI_01 : FB_MKS275;	
	
	{attribute 'pytmc' :=' pv : ST2K4:BCS:GCC:01 '}	
	{attribute 'TcLinkTo' := 	'.i_iPRESS_R	:=	TIIB[B940_K4S28_EB1 (EP3174-0002)]^AI Standard Channel 2^Value;
								 .q_xHV_DIS		:= 	TIIB[B940_K4S28_EB2 (EP2624-0002)]^Channel 1^Output	'}	
	ST2K4_BCS_GCC_01 : FB_MKS500_EP;		

						 
	{attribute 'pytmc' :=' pv : PC4K4:XTES:GPI:01 '}
	{attribute 'TcLinkTo' := 	'.i_iPRESS_R	:=	TIIB[B940_K4S33_EB2 (EP3174-0002)]^AI Standard Channel 1^Value	'}
	PC4K4_XTES_GPI_01 : FB_MKS275;

	{attribute 'pytmc' :=' pv : PC4K4:XTES:GCC:01 '}
	{attribute 'TcLinkTo' := 	'.i_iPRESS_R	:=	TIIB[B940_K4S33_EB2 (EP3174-0002)]^AI Standard Channel 2^Value;
								 .q_xHV_DIS		:= 	TIIB[B940_K4S33_EB3 (EP2624-0002)]^Channel 1^Output	'}	
	
	PC4K4_XTES_GCC_01 : FB_MKS500_EP;
	
	

	
(* Ion Pumps *)	
	
(*example
	{attribute 'TcLinkTo' := 	'.i_iPRESS		:=	TIIB[QPC_E1_EL3064]^AI Standard Channel 1^Value;
								 .i_xSP_DI		:= 	TIIB[QPC_E2_EL1004]^Channel 1^Input;
								 .q_xHVEna_DO	:= 	TIIB[QPC_E3_EL2794]^Channel 1^Output	'}
	{attribute 'pytmc' := '
		pv : RTDSL0:VAC:PIP:01
		io: io
	'}
	RTDSL0_PIP_01 : FB_PIP_Gamma;
	*)

	{attribute 'pytmc' :=' 
			pv : MR1K4:SOMS:PIP:01 '
 		}
	{attribute 'TcLinkTo' := 	'.i_iPRESS		:=	TIIB[CX0_E6_QPC1 (EL3064)]^AI Standard Channel 1^Value;
								 .i_xSP_DI		:= 	TIIB[CX0_E7_QPC1 (EL1004)]^Channel 1^Input;
								 .q_xHVEna_DO	:= 	TIIB[CX0_E8_QPC1 (EL2794)]^Channel 1^Output
	'}
	MR1K4_SOMS_PIP_01 : FB_PIP_Gamma;
	
	{attribute 'pytmc' :=' pv : ST1K4:TEST:PIP:01 '}
	{attribute 'TcLinkTo' := 	'.i_iPRESS		:=	TIIB[CX0_E6_QPC1 (EL3064)]^AI Standard Channel 2^Value;
								 .i_xSP_DI		:= 	TIIB[CX0_E7_QPC1 (EL1004)]^Channel 2^Input;
								 .q_xHVEna_DO	:= 	TIIB[CX0_E8_QPC1 (EL2794)]^Channel 2^Output
	'}	
	ST1K4_TEST_PIP_01 : FB_PIP_Gamma;	
	
	{attribute 'pytmc' :=' pv : ST2K4:BCS:PIP:01 '}
	{attribute 'TcLinkTo' := 	'.i_iPRESS		:=	TIIB[CX0_E6_QPC1 (EL3064)]^AI Standard Channel 3^Value;
								 .i_xSP_DI		:= 	TIIB[CX0_E7_QPC1 (EL1004)]^Channel 3^Input;
								 .q_xHVEna_DO	:= 	TIIB[CX0_E8_QPC1 (EL2794)]^Channel 3^Output
	'}
	ST2K4_BCS_PIP_01 : FB_PIP_Gamma;	

	{attribute 'pytmc' :=' pv : ST3K4:PPS:PIP:01 '}
	{attribute 'TcLinkTo' := 	'.i_iPRESS		:=	TIIB[CX0_E6_QPC1 (EL3064)]^AI Standard Channel 4^Value;
								 .i_xSP_DI		:= 	TIIB[CX0_E7_QPC1 (EL1004)]^Channel 4^Input;
								 .q_xHVEna_DO	:= 	TIIB[CX0_E8_QPC1 (EL2794)]^Channel 4^Output
	'}
	ST3K4_PPS_PIP_01 : FB_PIP_Gamma;		
	
	{attribute 'pytmc' :=' pv : PC4K4:XTES:PIP:01 '}
	{attribute 'TcLinkTo' := 	'.i_iPRESS		:=	TIIB[CX0_E9_QPC2 (EL3064)]^AI Standard Channel 1^Value;
								 .i_xSP_DI		:= 	TIIB[CX0_E10_QPC2 (EL1004)]^Channel 1^Input;
								 .q_xHVEna_DO	:= 	TIIB[CX0_E11_QPC2 (EL2794)]^Channel 1^Output
	'}
	PC4K4_XTES_PIP_01 : FB_PIP_Gamma;		

	
	
	

END_VAR

// ---- GVLs/GVL_FSV_PMPS.TcGVL
VAR_GLOBAL

	
	{'attribute 'pytmc' := 'pv: TMO:VAC:FFO:03  '}
    //{attribute 'TcLinkTo' := '.q_xFastFaultOut:=TIIB[CX0_E1 (EL2202)]^Channel 2^Output'}
    g_FastFaultOutput3  :   FB_HardwareFFOutput;	//FFO for TV1K4-VFS-1
	
	
END_VAR

// ---- GVLs/GVL_FS_Devices.TcGVL
VAR_GLOBAL

    {attribute 'pytmc' := '
		pv: TV1K4:VFS:01
	'}

	{attribute 'TcLinkTo' := 	'.q_xPress_OK		:= 	TIPC^PLC_TMO_VAC^PLC_TMO_VAC Instance^FSVTask Inputs^GVL_FS_Devices.TV1K4_VFS_1.i_xPress_OK;
								 .q_xOPN_SW			:=  TIPC^PLC_TMO_VAC^PLC_TMO_VAC Instance^FSVTask Inputs^GVL_FS_Devices.TV1K4_VFS_1.i_xOPN_SW;
								 .q_xCLS_SW			:=  TIPC^PLC_TMO_VAC^PLC_TMO_VAC Instance^FSVTask Inputs^GVL_FS_Devices.TV1K4_VFS_1.i_xCLS_SW;
								 .q_xVAC_FAULT_Reset:= 	TIPC^PLC_TMO_VAC^PLC_TMO_VAC Instance^FSVTask Inputs^GVL_FS_Devices.TV1K4_VFS_1.i_xVAC_FAULT_Reset;
								 .q_xOverrideMode	:= 	TIPC^PLC_TMO_VAC^PLC_TMO_VAC Instance^FSVTask Inputs^GVL_FS_Devices.TV1K4_VFS_1.i_xOverrideMode;
								 .q_xOverrideOpen	:= 	TIPC^PLC_TMO_VAC^PLC_TMO_VAC Instance^FSVTask Inputs^GVL_FS_Devices.TV1K4_VFS_1.i_xOverrideOpen;
								 .i_xTrigger		:=	TIPC^PLC_TMO_VAC^PLC_TMO_VAC Instance^FSVTask Outputs^GVL_FS_Devices.TV1K4_VFS_1.q_xTrigger
								 .i_xVFS_Open		:=	TIPC^PLC_TMO_VAC^PLC_TMO_VAC Instance^FSVTask Outputs^GVL_FS_Devices.TV1K4_VFS_1.q_xVFS_Open;
								 .i_xVFS_Closed		:=	TIPC^PLC_TMO_VAC^PLC_TMO_VAC Instance^FSVTask Outputs^GVL_FS_Devices.TV1K4_VFS_1.q_xVFS_Closed;
								 .i_xVAC_FAULT_OK	:=  TIPC^PLC_TMO_VAC^PLC_TMO_VAC Instance^FSVTask Outputs^GVL_FS_Devices.TV1K4_VFS_1.q_xVAC_FAULT_OK;
								 .i_xMPS_OK			:=  TIPC^PLC_TMO_VAC^PLC_TMO_VAC Instance^FSVTask Outputs^GVL_FS_Devices.TV1K4_VFS_1.q_xMPS_OK;
								 .i_eVFS_State		:=	TIPC^PLC_TMO_VAC^PLC_TMO_VAC Instance^FSVTask Outputs^GVL_FS_Devices.TV1K4_VFS_1.q_eVFS_State
	'}
	
	TV1K4_VFS_Interface : FB_VFS_Interface;


	{attribute 'TcLinkTo' := 	'
		.q_xClose_A	:=	TIIB[B940_K4S20_EK0  (EK1100)^K4S20-E2-FSV (EL2202)^Channel 1^Output;
		.q_xClose_B	:=	TIIB[B940_K4S20_EK0  (EK1100)^K4S20-E2-FSV (EL2202)^Channel 2^Output;
		.q_xClose_C	:=	TIIB[B940_K4S20_EK0  (EK1100)^K4S20-E3-FSV (EL2202)^Channel 1^Output;
		.q_xOPN_DO	:=	TIIB[B940_K4S20_EK0  (EK1100)^K4S20-E3-FSV (EL2202)^Channel 2^Output;
		.i_xClsLS	:=	TIIB[B940_K4S20_EK0  (EK1100)^K4S20-E1-FSV (EL1004)^Channel 1^Input;
		.i_xOpnLS	:=	TIIB[B940_K4S20_EK0  (EK1100)^K4S20-E1-FSV (EL1004)^Channel 2^Input;
		.i_xTrigger := 	TIIB[B940_R20_EK0 (EK1100)]^R20_EK0_E5_MKS937B (EL1124)^Channel 1^Input '}
	TV1K4_VFS_1 : FB_VFS;	
	
	
    {attribute 'pytmc' := '
		pv: MR3K4:KBO:VFS:01
	'}
	
	{attribute 'TcLinkTo' := 	'.q_xPress_OK		:= 	TIPC^PLC_TMO_VAC^PLC_TMO_VAC Instance^FSVTask Inputs^GVL_FS_Devices.MR3K4_KBO_VFS_1.i_xPress_OK;
								 .q_xOPN_SW			:=  TIPC^PLC_TMO_VAC^PLC_TMO_VAC Instance^FSVTask Inputs^GVL_FS_Devices.MR3K4_KBO_VFS_1.i_xOPN_SW;
								 .q_xCLS_SW			:=  TIPC^PLC_TMO_VAC^PLC_TMO_VAC Instance^FSVTask Inputs^GVL_FS_Devices.MR3K4_KBO_VFS_1.i_xCLS_SW;
								 .q_xVAC_FAULT_Reset:= 	TIPC^PLC_TMO_VAC^PLC_TMO_VAC Instance^FSVTask Inputs^GVL_FS_Devices.MR3K4_KBO_VFS_1.i_xVAC_FAULT_Reset;
								 .q_xOverrideMode	:= 	TIPC^PLC_TMO_VAC^PLC_TMO_VAC Instance^FSVTask Inputs^GVL_FS_Devices.MR3K4_KBO_VFS_1.i_xOverrideMode;
								 .q_xOverrideOpen	:= 	TIPC^PLC_TMO_VAC^PLC_TMO_VAC Instance^FSVTask Inputs^GVL_FS_Devices.MR3K4_KBO_VFS_1.i_xOverrideOpen;
								 .i_xTrigger		:=	TIPC^PLC_TMO_VAC^PLC_TMO_VAC Instance^FSVTask Outputs^GVL_FS_Devices.MR3K4_KBO_VFS_1.q_xTrigger
								 .i_xVFS_Open		:=	TIPC^PLC_TMO_VAC^PLC_TMO_VAC Instance^FSVTask Outputs^GVL_FS_Devices.MR3K4_KBO_VFS_1.q_xVFS_Open;
								 .i_xVFS_Closed		:=	TIPC^PLC_TMO_VAC^PLC_TMO_VAC Instance^FSVTask Outputs^GVL_FS_Devices.MR3K4_KBO_VFS_1.q_xVFS_Closed;
								 .i_xVAC_FAULT_OK	:=  TIPC^PLC_TMO_VAC^PLC_TMO_VAC Instance^FSVTask Outputs^GVL_FS_Devices.MR3K4_KBO_VFS_1.q_xVAC_FAULT_OK;
								 .i_xMPS_OK			:=  TIPC^PLC_TMO_VAC^PLC_TMO_VAC Instance^FSVTask Outputs^GVL_FS_Devices.MR3K4_KBO_VFS_1.q_xMPS_OK;
								 .i_eVFS_State		:=	TIPC^PLC_TMO_VAC^PLC_TMO_VAC Instance^FSVTask Outputs^GVL_FS_Devices.MR3K4_KBO_VFS_1.q_eVFS_State
	'}
	
	MR3K4_KBO_VFS_Interface : FB_VFS_Interface;	
	
	{attribute 'TcLinkTo' := 	'
		.q_xClose_A	:=	TIIB[K4S2_01_E3_VFS (EL2202)]^Channel 1^Output;
		.q_xClose_B	:=	TIIB[K4S2_01_E3_VFS (EL2202)]^Channel 2^Output;
		.q_xClose_C	:=	TIIB[K4S2_01_E4_VFS (EL2202)]^Channel 1^Output;
		.q_xOPN_DO	:=	TIIB[K4S2_01_E4_VFS (EL2202)]^Channel 2^Output;
		.i_xClsLS	:=	TIIB[K4S2_01_E1_VFS (EL1004)]^Channel 1^Input;
		.i_xOpnLS	:=	TIIB[K4S2_01_E1_VFS (EL1004)]^Channel 2^Input;
		.i_xTrigger :=  TIIB[B940_R20_EK0 (EK1100)]^R20_EK0_E5_MKS937B (EL1124)^Channel 1^Input'}
	MR3K4_KBO_VFS_1 : FB_VFS;
	
	{attribute 'pytmc' := '
		pv: MR3K4:KBO:VFS_1
	'}
	
	{attribute 'TcLinkTo' := 	'.q_xPress_OK		:= 	TIPC^PLC_TMO_VAC^PLC_TMO_VAC Instance^FSVTask Inputs^GVL_FS_Devices.MR4K4_KBO_VFS_1.i_xPress_OK;
								 .q_xOPN_SW			:=  TIPC^PLC_TMO_VAC^PLC_TMO_VAC Instance^FSVTask Inputs^GVL_FS_Devices.MR4K4_KBO_VFS_1.i_xOPN_SW;
								 .q_xCLS_SW			:=  TIPC^PLC_TMO_VAC^PLC_TMO_VAC Instance^FSVTask Inputs^GVL_FS_Devices.MR4K4_KBO_VFS_1.i_xCLS_SW;
								 .q_xVAC_FAULT_Reset:= 	TIPC^PLC_TMO_VAC^PLC_TMO_VAC Instance^FSVTask Inputs^GVL_FS_Devices.MR4K4_KBO_VFS_1.i_xVAC_FAULT_Reset;
								 .q_xOverrideMode	:= 	TIPC^PLC_TMO_VAC^PLC_TMO_VAC Instance^FSVTask Inputs^GVL_FS_Devices.MR4K4_KBO_VFS_1.i_xOverrideMode;
								 .q_xOverrideOpen	:= 	TIPC^PLC_TMO_VAC^PLC_TMO_VAC Instance^FSVTask Inputs^GVL_FS_Devices.MR4K4_KBO_VFS_1.i_xOverrideOpen;
								 .i_xTrigger		:=	TIPC^PLC_TMO_VAC^PLC_TMO_VAC Instance^FSVTask Outputs^GVL_FS_Devices.MR4K4_KBO_VFS_1.q_xTrigger
								 .i_xVFS_Open		:=	TIPC^PLC_TMO_VAC^PLC_TMO_VAC Instance^FSVTask Outputs^GVL_FS_Devices.MR4K4_KBO_VFS_1.q_xVFS_Open;
								 .i_xVFS_Closed		:=	TIPC^PLC_TMO_VAC^PLC_TMO_VAC Instance^FSVTask Outputs^GVL_FS_Devices.MR4K4_KBO_VFS_1.q_xVFS_Closed;
								 .i_xVAC_FAULT_OK	:=  TIPC^PLC_TMO_VAC^PLC_TMO_VAC Instance^FSVTask Outputs^GVL_FS_Devices.MR4K4_KBO_VFS_1.q_xVAC_FAULT_OK;
								 .i_xMPS_OK			:=  TIPC^PLC_TMO_VAC^PLC_TMO_VAC Instance^FSVTask Outputs^GVL_FS_Devices.MR4K4_KBO_VFS_1.q_xMPS_OK;
								 .i_eVFS_State		:=	TIPC^PLC_TMO_VAC^PLC_TMO_VAC Instance^FSVTask Outputs^GVL_FS_Devices.MR4K4_KBO_VFS_1.q_eVFS_State
	'}
	
	MR4K4_KBO_VFS_Interface : FB_VFS_Interface;	
	
	{attribute 'TcLinkTo' := 	'
		.q_xClose_A	:=	TIIB[K4S8_01_E3 (EL2202)]^Channel 1^Output;
		.q_xClose_B	:=	TIIB[K4S8_01_E3 (EL2202)]^Channel 2^Output;
		.q_xClose_C	:=	TIIB[K4S8_01_E4 (EL2202)]^Channel 1^Output;
		.q_xOPN_DO	:=	TIIB[K4S8_01_E4 (EL2202)]^Channel 2^Output;
		.i_xClsLS	:=	TIIB[K4S8_01_E1 (EL1004)]^Channel 1^Input;
		.i_xOpnLS	:=	TIIB[K4S8_01_E1 (EL1004)]^Channel 2^Input;
		.i_xTrigger := 	TIIB[B940_R20_EK0 (EK1100)]^R20_EK0_E5_MKS937B (EL1124)^Channel 1^Input '}
	MR4K4_KBO_VFS_1 : FB_VFS;
END_VAR

// ---- GVLs/GVL_Hutch_Gauges.TcGVL
//{attribute 'qualified_only'}
VAR_GLOBAL
(* Pirani & Cold Cathode*)

	{attribute 'pytmc' :=' pv: MR2K4:KBO:GPI:01 '}
	{attribute 'TcLinkTo' := 	'.i_iPRESS_R	:=	TIIB[TMO_K4S2_DRL_02 (EK1100)]^K4S2_02_E1 (EL3174)^AI Standard Channel 2^Value '}
	MR2K4_KBO_GPI_01 : FB_MKS275;
	
	{attribute 'pytmc' :=' pv: MR2K4:KBO:GCC:01 '}
	{attribute 'TcLinkTo' := 	'.i_iPRESS_R	:=	TIIB[TMO_K4S2_DRL_02 (EK1100)]^K4S2_02_E1 (EL3174)^AI Standard Channel 3^Value;
								 .i_xHV_ON	    :=	TIIB[TMO_K4S2_DRL_02 (EK1100)]^K4S2_02_E7 (EL1124)^Channel 3^Input;
								 .i_xDisc_Active:=	TIIB[TMO_K4S2_DRL_02 (EK1100)]^K4S2_02_E7 (EL1124)^Channel 4^Input;								 
								 .q_xHV_DIS		:= 	TIIB[TMO_K4S2_DRL_02 (EK1100)]^K4S2_02_E5 (EL2624)^Channel 2^Output	'}	
	MR2K4_KBO_GCC_01 : FB_MKS500;
	
	{attribute 'pytmc' :=' pv: PA1K4:IP1:GPI:01 '}
	{attribute 'TcLinkTo' := 	'.i_iPRESS_R	:=	TIIB[TMO_K4S2_DRL_02 (EK1100)]^K4S2_02_E2 (EL3174)^AI Standard Channel 1^Value '}	
	PA1K4_IP1_GPI_01 : FB_MKS275;
	

	{attribute 'pytmc' :=' pv: PA1K4:IP1:GCC:01 '}
	{attribute 'TcLinkTo' := 	'.i_iPRESS_R	:=	TIIB[TMO_K4S2_DRL_02 (EK1100)]^K4S2_02_E1 (EL3174)^AI Standard Channel 4^Value;
								 .i_xHV_ON	    :=	TIIB[TMO_K4S2_DRL_02 (EK1100)]^K4S2_02_E8 (EL1124)^Channel 1^Input;
								 .i_xDisc_Active:=	TIIB[TMO_K4S2_DRL_02 (EK1100)]^K4S2_02_E8 (EL1124)^Channel 2^Input;								 
								 .q_xHV_DIS		:= 	TIIB[TMO_K4S2_DRL_02 (EK1100)]^K4S2_02_E5 (EL2624)^Channel 3^Output	'}		
	PA1K4_IP1_GCC_01 : FB_MKS500;
	

	{attribute 'pytmc' :=' pv: IM4K4:PPM:GCC:01 '}
	{attribute 'TcLinkTo' := 	'.i_iPRESS_R	:=	TIIB[TMO_K4S2_DRL_02 (EK1100)]^K4S2_02_E2 (EL3174)^AI Standard Channel 2^Value;
								 .i_xHV_ON	    :=	TIIB[TMO_K4S2_DRL_02 (EK1100)]^K4S2_02_E8 (EL1124)^Channel 3^Input;
								 .i_xDisc_Active:=	TIIB[TMO_K4S2_DRL_02 (EK1100)]^K4S2_02_E8 (EL1124)^Channel 4^Input;								 
								 .q_xHV_DIS		:= 	TIIB[TMO_K4S2_DRL_02 (EK1100)]^K4S2_02_E5 (EL2624)^Channel 4^Output	'}			
	IM4K4_PPM_GCC_01 : FB_MKS500;
	
	
	{attribute 'pytmc' := '	pv: LI2K4:IP1:GFS:01
		io: io
	'}
	{attribute 'TcLinkTo' := 	'.i_iPRESS_R	:=	TIIB[^B940_R20_EK0 (EK1100)]^R20_EK0_E1_MKS937B (EL3064)^AI Standard Channel 1^Value;
								 .q_xHV_DIS		:= 	TIIB[^B940_R20_EK0 (EK1100)]^R20_EK0_E3_MKS937B (EL2794)^Channel 1^Output
	'}
    LI2K4_IP1_GFS_01 : FB_MKS422;
	
	
	{attribute 'pytmc' :=' pv: TM1K4:GCC:01 '}
	{attribute 'TcLinkTo' := 	'.i_iPRESS_R	:=	TIIB[TMO_K4S6_DRL_01 (EK1100)]^K4S6_01_E15 (EL3174)^AI Standard Channel 1^Value;
								 .i_xHV_ON	    :=	TIIB[TMO_K4S6_DRL_01 (EK1100)]^K4S6_01_E20 (EL1124)^Channel 1^Input;
								 .i_xDisc_Active:=	TIIB[TMO_K4S6_DRL_01 (EK1100)]^K4S6_01_E20 (EL1124)^Channel 2^Input;								 
								 .q_xHV_DIS		:= 	TIIB[TMO_K4S6_DRL_01 (EK1100)]^K4S6_01_E14 (EL2624)^Channel 1^Output	'}		
	TM1K4_GCC_01 : FB_MKS500;
	
	{attribute 'pytmc' :=' pv: IM5K4:PPM:GCC:01 '}
	{attribute 'TcLinkTo' := 	'.i_iPRESS_R	:=	TIIB[TMO_K4S6_DRL_01 (EK1100)]^K4S6_01_E15 (EL3174)^AI Standard Channel 2^Value;
								 .i_xHV_ON	    :=	TIIB[TMO_K4S6_DRL_01 (EK1100)]^K4S6_01_E20 (EL1124)^Channel 3^Input;
								 .i_xDisc_Active:=	TIIB[TMO_K4S6_DRL_01 (EK1100)]^K4S6_01_E20 (EL1124)^Channel 4^Input;								 
								 .q_xHV_DIS		:= 	TIIB[TMO_K4S6_DRL_01 (EK1100)]^K4S6_01_E14 (EL2624)^Channel 2^Output	'}		
	IM5K4_PPM_GCC_01 : FB_MKS500;
	
	
	{attribute 'pytmc' :=' pv: PA2K4:IP1:GPI:01 '}
	{attribute 'TcLinkTo' := 	'.i_iPRESS_R	:=	TIIB[TMO_K4S6_DRL_01 (EK1100)]^K4S6_01_E15 (EL3174)^AI Standard Channel 4^Value '}	
	PA2K4_IP1_GPI_01 : FB_MKS275;
	
	{attribute 'pytmc' :=' pv: PA2K4:IP1:GCC:01 '}
	{attribute 'TcLinkTo' := 	'.i_iPRESS_R	:=	TIIB[TMO_K4S6_DRL_01 (EK1100)]^K4S6_01_E15 (EL3174)^AI Standard Channel 3^Value;
								 .i_xHV_ON	    :=	TIIB[TMO_K4S6_DRL_01 (EK1100)]^K4S6_01_E21 (EL1124)^Channel 1^Input;
								 .i_xDisc_Active:=	TIIB[TMO_K4S6_DRL_01 (EK1100)]^K4S6_01_E21 (EL1124)^Channel 2^Input;								 
								 .q_xHV_DIS		:= 	TIIB[TMO_K4S6_DRL_01 (EK1100)]^K4S6_01_E14 (EL2624)^Channel 3^Output	'}		
	PA2K4_IP1_GCC_01 : FB_MKS500;


	{attribute 'pytmc' :=' pv: MR4K4:KBO:GPI:01 '}
	{attribute 'TcLinkTo' := 	'.i_iPRESS_R	:=	TIIB[TMO_K4S6_DRL_01 (EK1100)]^K4S6_01_E18 (EL3174)^AI Standard Channel 1^Value '}		
	MR4K4_KBO_GPI_01 : FB_MKS275;

	{attribute 'pytmc' :=' pv: MR4K4:KBO:GCC:01 '}
	{attribute 'TcLinkTo' := 	'.i_iPRESS_R	:=	TIIB[TMO_K4S6_DRL_01 (EK1100)]^K4S6_01_E18 (EL3174)^AI Standard Channel 2^Value;
								 .i_xHV_ON	    :=	TIIB[TMO_K4S6_DRL_01 (EK1100)]^K4S6_01_E21 (EL1124)^Channel 3^Input;
								 .i_xDisc_Active:=	TIIB[TMO_K4S6_DRL_01 (EK1100)]^K4S6_01_E21 (EL1124)^Channel 4^Input;								 
								 .q_xHV_DIS		:= 	TIIB[TMO_K4S6_DRL_01 (EK1100)]^K4S6_01_E14 (EL2624)^Channel 4^Output	'}			
	MR4K4_KBO_GCC_01 : FB_MKS500;
	
	(* Roughing gauges *)

	{attribute 'pytmc' :=' pv: TMO:ROUGH1:GPI:01 '}
	{attribute 'TcLinkTo' := 	'.i_iPRESS_R	:=	TIIB[TMO_WALL_WEST_EP01 (EP4374-0002)]^AI Inputs Channel 1^Value	'}	
	TMO_ROUGH1_GPI_01 : FB_9XX;
	
	{attribute 'pytmc' :=' pv: TMO:ROUGH1:GPI:02 '}
	{attribute 'TcLinkTo' := 	'.i_iPRESS_R	:=	TIIB[TMO_K4S2_ EP1 (EP4374-0002)]^AI Inputs Channel 1^Value	'}	
	TMO_ROUGH1_GPI_02 : FB_9XX;
	
	{attribute 'pytmc' :=' pv: TMO:ROUGH1:GPI:03 '}
	{attribute 'TcLinkTo' := 	'.i_iPRESS_R	:=	TIIB[TMO_K4S6_ EP1 (EP4374-0002)]^AI Inputs Channel 1^Value	'}		
	TMO_ROUGH1_GPI_03 : FB_9XX;

	{attribute 'pytmc' :=' pv: TMO:ROUGH2:GPI:01 '}
	{attribute 'TcLinkTo' := 	'.i_iPRESS_R	:=	TIIB[TMO_WALL_WEST_EP01 (EP4374-0002)]^AI Inputs Channel 2^Value	'}	
	TMO_ROUGH2_GPI_01 : FB_9XX;
	
	{attribute 'pytmc' :=' pv: TMO:ROUGH2:GPI:02 '}
	{attribute 'TcLinkTo' := 	'.i_iPRESS_R	:=	TIIB[TMO_K4S2_ EP1 (EP4374-0002)]^AI Inputs Channel 2^Value	'}	
	TMO_ROUGH2_GPI_02 : FB_9XX;	
	
	
	

END_VAR

// ---- GVLs/GVL_PMPS.TcGVL
//{attribute 'qualified_only'}
VAR_GLOBAL
	
//Example implementation of the FFO
    {attribute 'pytmc' := '
    {pv: TMO:VAC:FFO:01    '}
    {attribute 'TcLinkTo' := '.q_xFastFaultOut:=TIIB[CX0_E1 (EL2202)]^Channel 1^Output'}
    g_FastFaultOutput1  :   FB_HardwareFFOutput;	//FFO for ST3K4_PPS's Upstream Components
	
	 {attribute 'pytmc' := 'pv: TMO:VAC:FFO:02  '}
    {attribute 'TcLinkTo' := '.q_xFastFaultOut:=TIIB[CX0_E1 (EL2202)]^Channel 2^Output'}
    g_FastFaultOutput2  :   FB_HardwareFFOutput;	//FFO for ST3K4_PPS's Downstream Components
	
	
	
	 {attribute 'pytmc' := 'pv: TMO:VAC:FFO:04  '}
   // {attribute 'TcLinkTo' := '.q_xFastFaultOut:=TIIB[CX0_E1 (EL2202)]^Channel 2^Output'}
    g_FastFaultOutput4  :   FB_HardwareFFOutput;
	
	{attribute 'pytmc' := '    'pv: PLC:TMO:VAC:RESET:FF1    '}
	xReset_PMPS_FFO1	:	BOOL	:=	FALSE;		//FFO RESET for ST3K4_PPS's Upstream Components
	{attribute 'pytmc' := '    pv: PLC:TMO:VAC:RESET:FF2  '}
	xReset_PMPS_FFO2	:	BOOL	:=	FALSE;		//FFO RESET for ST3K4_PPS's Downstream Components
	
	{attribute 'pytmc' := '
        pv: @(PREFIX)Arbiter:01
    '}
    g_fbArbiter1    :   FB_Arbiter(1);
	
	xTMO_FEE_MPS_OK: BOOL := TRUE;
	
	xTMO_NEH_MPS_OK: BOOL := TRUE;

END_VAR

// ---- GVLs/GVL_Variables.TcGVL
//{attribute 'qualified_only'}
VAR_GLOBAL
	
//	r_Accelerator_Setpoint	: REAL := 1E-12; (*unrealistic setpoint currently*)
	{attribute 'pytmc' := 'pv: TMO:FEE:VAC:OVRDON'}
	xSystemOverrideMode_FEE	: BOOL := FALSE; (* Global system override for the TMO FEE Vacuum System *)
	
	{attribute 'pytmc' := 'pv: TMO:NEH:VAC:OVRDON'}
	xSystemOverrideMode_TMO	: BOOL := FALSE; (* Global system override for the TMO hutch Vacuum System *)
END_VAR

// ---- POUs/DIAGNOSTICS.TcPOU
PROGRAM DIAGNOSTICS
VAR
	//Change the PLC String Name to the actual PLC NAME
	sPLCName :STRING := 'PLC-TMO-VAC';
	//Link the sAMSNetID to the Etherat Master netID
	i_sAMSNetID AT %I*: AMSNETID;
	// DO NOT CHANGE
	sAMSNetID : STRING; //used for EPICS PV
	sLibVersion_LCLS_General : STRING;(* := stLibVersion_LCLS_General.sVersion*) ;
	
	fbEcatDiag:FB_EcatDiag;
	{attribute 'pytmc' := ' pv: PLC:TMO:VAC:AllSlaveStateGood '}
	bAllSlaveStateGood : BOOL;
	{attribute 'pytmc' := ' pv: PLC:TMO:VAC:MasterStateGood '}	
	bMasterStateGood :BOOL;
	iMasterState: WORD;
	sMasterState:STRING;
	nSlaveNumber : UINT;
	aiSlaveStates: ARRAY[1..256] OF BYTE;
	aEcSlaveInfo :  ARRAY[1..256] OF ST_EcDevice;
END_VAR

// Instaniating a call to the fbEcatDiag
fbEcatDiag(
	I_AMSNetId:=i_sAMSNetID , 
	i_xFirstPass:= _TaskInfo[1].FirstCycle, 
	q_xAllSlaveStatesGood=> bAllSlaveStateGood , 
	q_anTermStates=> aiSlaveStates, 
	q_xMasterStateGood=>bMasterStateGood , 
	q_nMasterState=> iMasterState, 
	q_sMasterState=> sMasterState , 
	q_astEcConfSlaveInfo=> aEcSlaveInfo , 
	q_nSlaves=> nSlaveNumber);

END_PROGRAM

// ---- POUs/MAIN.TcPOU
PROGRAM MAIN
VAR

	fbLogHandler : FB_LogHandler;
	
END_VAR


fbLogHandler();

// Run the Diagnostics PRG
DIAGNOSTICS();

(* FEE devices*)
PRG_FEE();
PMPS();

(*Hutch*)
PRG_Hutch_Gauges();
PRG_Hutch_Beamline_Valves();
PRG_Roughing_Pumps();

END_PROGRAM

// ---- POUs/PRG_FEE.TcPOU
 PROGRAM PRG_FEE
VAR
ADS_connection_counter : UDINT;	

(*Upstream Interface*)
	
    USG_PIP : ST_VG;
	
	USG_VGC : ST_VG;


END_VAR

(* Gauges*)
   (* Read GCC from upstream PLC - plc-kfe-vac*)
  (* MR1K4_GCC_01_ADS(
	sNetId:= '172.21.92.61.1.1', 
	nPort:=851 , 
	sVarName:= 'fb_MR1K4_SOMS_GCC_1' , 
	iWatchdog:=ADS_connection_counter , 
	IG=> , 
	bError=> ); *)
	(* if upstream vacuum ok, set upstream press at good levels *)  
    IF USVacOk_HI THEN 
		USG_VGC.xAT_VAC := TRUE;
		USG_VGC.rPRESS := 5E-7;
		USG_VGC.xPRESS_OK := TRUE;
	ELSE
		USG_VGC.xPRESS_OK := FALSE;
		USG_VGC.xAT_VAC := FALSE;
	END_IF

    IF USVacOk_LO THEN 
		USG_PIP.rPRESS := 5E-5;
		USG_PIP.xPRESS_OK := TRUE;
		USG_PIP.xAT_VAC := TRUE;
	ELSE
		USG_PIP.xPRESS_OK := FALSE;
		USG_PIP.xAT_VAC := FALSE;
	END_IF 

	(* check other gauges*)
	TV1K4_GPI_01(); 
	ST1K4_TEST_GPI_01(); 
	ST2K4_BCS_GPI_01();
	PC4K4_XTES_GPI_01(); 
	
	TV1k4_GCC_01(PG:=TV1k4_GPI_01.PG , IG=> );
	ST1K4_TEST_GCC_01(PG:=ST1K4_TEST_GPI_01.PG , IG=> ); 
	ST2K4_BCS_GCC_01(PG:=ST2K4_BCS_GPI_01.PG , IG=> );
	PC4K4_XTES_GCC_01(PG:=PC4K4_XTES_GPI_01.PG , IG=> );
		
(* Valves*)
(*example
GEM1_VGC_10(i_stUSG := USG_GCC.IG, i_stDSG:= GEM1_GCC_10.IG,i_xDis_DPIlk := TRUE, i_xEPS_OK := TRUE,
		i_xPMPS_OK := TRUE, i_xExt_OK := xGEM1_AperturesOpnOK, i_xOverrideMode := xGEM1OverrideMode,i_xReset := xFastFaultReset,io_fbFFHWO :=g_FastFaultOutput1);
*)
	TV1K4_VGC_01(
				i_stUSG := USG_VGC, 
				i_stDSG:= TV1k4_GCC_01.IG, 
				i_xDis_DPIlk := FALSE, 
				i_xEPS_OK := TRUE,
				i_xPMPS_OK := TRUE, 
				i_xExt_OK := TRUE, 
				i_xOverrideMode := xSystemOverrideMode_FEE, 
				i_xReset := xReset_PMPS_FFO1,
				io_fbFFHWO :=g_FastFaultOutput1,
				fbArbiter := g_fbArbiter1);
	
 	TV1K4_VGC_02(
				i_stUSG := TV1k4_GCC_01.IG, 
				i_stDSG:= ST1K4_TEST_GCC_01.IG, 
				i_xDis_DPIlk := FALSE, 
				i_xEPS_OK := TRUE,
				i_xPMPS_OK := TRUE, 
				i_xExt_OK := TRUE, 
				i_xOverrideMode := xSystemOverrideMode_FEE, 
				i_xReset := xReset_PMPS_FFO1,
				io_fbFFHWO :=g_FastFaultOutput1,
                fbArbiter := g_fbArbiter1);
	
	ST3K4_PPS_VGC_01(
				i_stUSG := ST2K4_BCS_GCC_01.IG, 
				i_stDSG:= PC4K4_XTES_GCC_01.IG, 
				i_xDis_DPIlk := FALSE, 
				i_xEPS_OK := TRUE,
				i_xPMPS_OK := TRUE, 
				i_xExt_OK := TRUE, 
				i_xOverrideMode := xSystemOverrideMode_FEE, 
				i_xReset := xReset_PMPS_FFO2,
				io_fbFFHWO :=g_FastFaultOutput2,
                fbArbiter := g_fbArbiter1);
				
(*Ion Pumps*)	
	(*example
	SP1L0_KMONO_PIP_01(i_stGauge:=SP1L0_KMONO_GCC_01.IG, stPump=>);*)		

	MR1K4_SOMS_PIP_01(i_stGauge := USG_PIP, stPump=>);
	ST1K4_TEST_PIP_01(i_stGauge := ST1K4_TEST_GCC_01.IG, stPump=>);
	ST2K4_BCS_PIP_01(i_stGauge := ST2K4_BCS_GCC_01.IG, stPump=>);
	ST3K4_PPS_PIP_01(i_stGauge := ST2K4_BCS_GCC_01.IG, stPump=>);
	PC4K4_XTES_PIP_01(i_stGauge := PC4K4_XTES_GCC_01.IG, stPump=>);

END_PROGRAM

// ---- POUs/PMPS.TcPOU
PROGRAM PMPS
VAR
	
END_VAR

(*FastFaultOuput*)
g_FastFaultOutput1.Execute(bAutoReset:= TRUE);
g_FastFaultOutput2.Execute(i_xVeto:=PMPS_GVL.stCurrentBeamParameters.aStoppers[K_Stopper.ST1], bAutoReset:= TRUE);

END_PROGRAM

// ---- POUs/PRG_Roughing_Pumps.TcPOU
PROGRAM PRG_Roughing_Pumps
VAR
	
	xRough1Vrc01_OpenOK: BOOL := False;
	xRough1Vrc02_OpenOK: BOOL := False;
	xRough2Vrc01_OpenOK: BOOL := False;
	dummy_FFFO : FB_HardwareFFOutput;
	dummy_fbArbiter1    :   FB_Arbiter(1);
	
	PA1K4_IP1_PTM_01_xExtIlkOK: BOOL := FALSE;
	PA1K4_IP1_PTM_02_xExtIlkOK: BOOL := FALSE;
	PA1K4_IP1_PTM_03_xExtIlkOK: BOOL := False;
	
	

	tonDelOK : TON;
	tDelOK	:	TIME := T#30S;
	xExtIlkOK : BOOL;
	
	
	
	
	IM4K4_PPM_PTM_01_xExtIlkOK: BOOL := FALSE;
	LI1K4_IP1_PTM_01_xExtIlkOK: BOOL := FALSE;
	LI3K4_IP1_OUT_PTM_01_xExtIlkOK: BOOL := False;
	IM5K4_PPM_PTM_01_xExtIlkOK: BOOL := False;
	
	rTolerance : REAL;
	xDifPressureOK : BOOL := FALSE;
	TMO_ROUGH1_VRC_01_xExt_OK : BOOL;
	TMO_ROUGH1_VRC_02_xExt_OK : BOOL;
	
END_VAR

VAR RETAIN
	TM1K4_PTM_01_xExtIlkOK: BOOL := False;
END_VAR


(* Roughing Valves *)

(* All three roughing valves permit to open when both side reading pressure below than setpoint, 1E-3 for both sides.
   When chamber is vented, bypass to open valve to pump down. 
   FB_VGC_2S is used for VRC controls.
   
   For TMO_ROUGH1_VRC_01 & TMO_ROUGH1_VRC_02, additional interlock is implemented using i_xExt_OK input of VGC function:
   If pressure difference between TMO_ROUGH1_GPI_02 and TMO_ROUGH1_GPI_03 is greater than 20 Torr, 
   only one of them permit to open.
   
*)


(* Check the pressure difference between TMO_ROUGH1_GPI_02 and TMO_ROUGH1_GPI_03 *) 



rTolerance := 0.1;
xDifPressureOK := (ABS(TMO_ROUGH1_GPI_02.PG.rPRESS - TMO_ROUGH1_GPI_03.PG.rPRESS ) <= rTolerance ) AND
				  TMO_ROUGH1_GPI_02.PG.xPRESS_OK AND TMO_ROUGH1_GPI_03.PG.xPRESS_OK;
				  
(* Set external interlock OK TRUE, when xDifPressureOK or TMO_ROUGH1_VRC_02 is closed *)				  
TMO_ROUGH1_VRC_01_xExt_OK := xDifPressureOK OR TMO_ROUGH1_VRC_02.iq_stValve.i_xClsLS; 
TMO_ROUGH1_VRC_02_xExt_OK := xDifPressureOK OR TMO_ROUGH1_VRC_01.iq_stValve.i_xClsLS; 


TMO_ROUGH1_VRC_01(
				i_stUSG := TMO_ROUGH1_GPI_02.PG, 
				i_stDSG:= TMO_ROUGH1_GPI_01.PG, 
				i_xDis_DPIlk := FALSE, 
				i_xEPS_OK := TRUE,
				i_xPMPS_OK := TRUE, 
				i_xExt_OK := TMO_ROUGH1_VRC_01_xExt_OK, 
				i_xOverrideMode := xSystemOverrideMode_TMO AND TMO_ROUGH1_VRC_01_xExt_OK,
				i_xReset := False,
				io_fbFFHWO :=dummy_FFFO,
                fbArbiter := dummy_fbArbiter1,
);


TMO_ROUGH1_VRC_02(
				i_stUSG := TMO_ROUGH1_GPI_03.PG, 
				i_stDSG:= TMO_ROUGH1_GPI_01.PG, 
				i_xDis_DPIlk := FALSE, 
				i_xEPS_OK := TRUE,
				i_xPMPS_OK := TRUE, 
				i_xExt_OK := TMO_ROUGH1_VRC_02_xExt_OK, 
				i_xOverrideMode := xSystemOverrideMode_TMO AND TMO_ROUGH1_VRC_02_xExt_OK, 
				i_xReset := false,
				io_fbFFHWO :=dummy_FFFO,
                fbArbiter := dummy_fbArbiter1);


TMO_ROUGH2_VRC_01(
				i_stUSG := TMO_ROUGH2_GPI_02.PG, 
				i_stDSG:= TMO_ROUGH2_GPI_01.PG, 
				i_xDis_DPIlk := FALSE, 
				i_xEPS_OK := TRUE,
				i_xPMPS_OK := TRUE, 
				i_xExt_OK := TRUE, 
				i_xOverrideMode := xSystemOverrideMode_TMO, 
				i_xReset := false,
				io_fbFFHWO :=dummy_FFFO,
                fbArbiter := dummy_fbArbiter1);


(* Granite 1 K4S2 Differential Turbo pumps *)


(* check if PA1K4_IP1_PTM_03 is Atspd, if it is starting, set up a timer for 30s to *)

xExtIlkOK := F_Turbo_Protection_ILK(i_stTurbo := PA1K4_IP1_PTM_01.iq_stPTM, 
			i_stISG := PA1K4_IP1_GPI_01.PG, 
			i_stBSG := TMO_ROUGH1_GPI_02.PG, 
			iq_stValve := TMO_ROUGH1_VRC_01.iq_stValve)	;
					
(* delay 30s to start if PTM03 is not at speed*)
IF (PA1K4_IP1_PTM_03.iq_stPTM.i_xAtSpd) AND (NOT PA1K4_IP1_PTM_03.iq_stPTM.i_xFault) THEN
		PA1K4_IP1_PTM_01_xExtIlkOK := xExtIlkOK;

ELSIF (PA1K4_IP1_PTM_03.iq_stPTM.q_RunDO ) AND (NOT PA1K4_IP1_PTM_03.iq_stPTM.i_xFault ) THEN
	//delay timer
  	  tonDelOK(IN:= xExtIlkOK, PT:=tDelOK);
	PA1K4_IP1_PTM_01_xExtIlkOK := xExtIlkOK AND tonDelOK.Q;	
ELSE
		PA1K4_IP1_PTM_01_xExtIlkOK := FALSE;			
END_IF


xExtIlkOK := F_Turbo_Protection_ILK(i_stTurbo := PA1K4_IP1_PTM_02.iq_stPTM, 
			i_stISG := PA1K4_IP1_GPI_01.PG, 
			i_stBSG := TMO_ROUGH1_GPI_02.PG, 
			iq_stValve := TMO_ROUGH1_VRC_01.iq_stValve)	;

IF (PA1K4_IP1_PTM_03.iq_stPTM.i_xAtSpd) AND (NOT PA1K4_IP1_PTM_03.iq_stPTM.i_xFault) THEN
		PA1K4_IP1_PTM_02_xExtIlkOK := xExtIlkOK;

ELSIF (PA1K4_IP1_PTM_03.iq_stPTM.q_RunDO ) AND (NOT PA1K4_IP1_PTM_03.iq_stPTM.i_xFault ) THEN
	//delay timer
  	  tonDelOK(IN:= xExtIlkOK, PT:=tDelOK);
	PA1K4_IP1_PTM_02_xExtIlkOK := xExtIlkOK AND tonDelOK.Q;	
ELSE
		PA1K4_IP1_PTM_02_xExtIlkOK := FALSE;			
END_IF

PA1K4_IP1_PTM_03_xExtIlkOK  := F_Turbo_Protection_ILK(i_stTurbo := PA1K4_IP1_PTM_03.iq_stPTM, 
			i_stISG := PA1K4_IP1_GPI_01.PG, 
			i_stBSG := TMO_ROUGH1_GPI_02.PG, 
			iq_stValve := TMO_ROUGH1_VRC_01.iq_stValve)	;


PA1K4_IP1_PTM_01(i_xExtIlkOK := PA1K4_IP1_PTM_01_xExtIlkOK , iq_stPTM => );

PA1K4_IP1_PTM_02(i_xExtIlkOK := PA1K4_IP1_PTM_02_xExtIlkOK, iq_stPTM => );
PA1K4_IP1_PTM_03(i_xExtIlkOK := PA1K4_IP1_PTM_03_xExtIlkOK, iq_stPTM => );

(*Serial Interface*)
(*Assign adresses to the pfeiffer controllers connected to this serial terminal*)
st_Pfeiffer_CTRL_PTM_01_02_03[1].iSerialAddress :=10;//PA1K4_IP1_PTM_01
st_Pfeiffer_CTRL_PTM_01_02_03[1].xEnableComm := TRUE;
st_Pfeiffer_CTRL_PTM_01_02_03[2].iSerialAddress :=9;//PA1K4_IP1_PTM_02
st_Pfeiffer_CTRL_PTM_01_02_03[2].xEnableComm := TRUE;
st_Pfeiffer_CTRL_PTM_01_02_03[3].iSerialAddress :=1;//PA1K4_IP1_PTM_03
st_Pfeiffer_CTRL_PTM_01_02_03[3].xEnableComm := TRUE;	
(* Instanitate the Function block for serial communication with Pfeiffer*)	
PA1K4_IP1_PTM_01_02_03_COM(astPfeifferControl := st_Pfeiffer_CTRL_PTM_01_02_03,
			   astPfeifferStatus:= st_Pfeiffer_RBK_PTM_01_02_03,
				SerialRXBuffer:= K4S2_02_E10_SerialRXBuffer,
				SerialTXBuffer:= K4S2_02_E10_SerialTXBuffer);
(* Copy Status Pv's into the PTM structure*)
PA1K4_IP1_PTM_01.M_Serial_IO(st_Pfeiffer_CTRL:=st_Pfeiffer_CTRL_PTM_01_02_03[1],st_Pfeiffer_RBK:=st_Pfeiffer_RBK_PTM_01_02_03[1]);				
PA1K4_IP1_PTM_02.M_Serial_IO(st_Pfeiffer_CTRL:=st_Pfeiffer_CTRL_PTM_01_02_03[2],st_Pfeiffer_RBK:=st_Pfeiffer_RBK_PTM_01_02_03[2]);				
PA1K4_IP1_PTM_03.M_Serial_IO(st_Pfeiffer_CTRL:=st_Pfeiffer_CTRL_PTM_01_02_03[3],st_Pfeiffer_RBK:=st_Pfeiffer_RBK_PTM_01_02_03[3]);				
		
(* Leybold turbo pumps on Granite 1 *)

IM4K4_PPM_PTM_01_xExtIlkOK := F_Turbo_Protection_ILK(i_stTurbo := IM4K4_PPM_PTM_01.iq_stPTM, 
			i_stISG := PA1K4_IP1_GPI_01.PG, 
			i_stBSG := TMO_ROUGH1_GPI_02.PG, 
			iq_stValve := TMO_ROUGH1_VRC_01.iq_stValve)	;

IM4K4_PPM_PTM_01(i_xExtIlkOK := IM4K4_PPM_PTM_01_xExtIlkOK, iq_stPTM => );

(* Instanitate the Function block for serial communication with TD20 *)
IM4K4_PPM_PTM_01_COM(SerialRXBuffer := K4S2_02_E17_SerialRXBuffer, 
				SerialTXBuffer:= K4S2_02_E17_SerialTXBuffer,
				astTD20Status=>);
(* Copy Status Pv's into the PTM structure*)
IM4K4_PPM_PTM_01.M_Serial_IO(IM4K4_PPM_PTM_01_COM.astTD20Status);



LI1K4_IP1_PTM_01_xExtIlkOK := F_Turbo_Protection_ILK(i_stTurbo := LI1K4_IP1_PTM_01.iq_stPTM, 
			i_stISG := PA1K4_IP1_GPI_01.PG, 
			i_stBSG := TMO_ROUGH1_GPI_02.PG, 
			iq_stValve := TMO_ROUGH1_VRC_01.iq_stValve)	;
			
LI1K4_IP1_PTM_01(i_xExtIlkOK := LI1K4_IP1_PTM_01_xExtIlkOK, iq_stPTM => );

(* Instanitate the Function block for serial communication with TD20 *)
LI1K4_IP1_PTM_01_COM(SerialRXBuffer := K4S2_02_E18_SerialRXBuffer, 
				SerialTXBuffer:= K4S2_02_E18_SerialTXBuffer,
				astTD20Status=>);
(* Copy Status Pv's into the PTM structure*)
LI1K4_IP1_PTM_01.M_Serial_IO(LI1K4_IP1_PTM_01_COM.astTD20Status);



(* Granite 2 K4S6 *)

LI3K4_IP1_OUT_PTM_01_xExtIlkOK := F_Turbo_Protection_ILK(i_stTurbo := LI3K4_IP1_OUT_PTM_01.iq_stPTM, 
			i_stISG := PA2K4_IP1_GPI_01.PG, 
			i_stBSG := TMO_ROUGH1_GPI_03.PG, 
			iq_stValve := TMO_ROUGH1_VRC_02.iq_stValve)	;

LI3K4_IP1_OUT_PTM_01(i_xExtIlkOK := LI3K4_IP1_OUT_PTM_01_xExtIlkOK, iq_stPTM => );

TM1K4_PTM_01_xExtIlkOK := F_Turbo_Protection_ILK(i_stTurbo := TM1K4_PTM_01.iq_stPTM, 
			i_stISG := PA2K4_IP1_GPI_01.PG, 
			i_stBSG := TMO_ROUGH1_GPI_03.PG, 
			iq_stValve := TMO_ROUGH1_VRC_02.iq_stValve)	;

TM1K4_PTM_01(i_xExtIlkOK := TM1K4_PTM_01_xExtIlkOK, iq_stPTM => );

IM5K4_PPM_PTM_01_xExtIlkOK := F_Turbo_Protection_ILK(i_stTurbo := IM5K4_PPM_PTM_01.iq_stPTM, 
			i_stISG := PA2K4_IP1_GPI_01.PG, 
			i_stBSG := TMO_ROUGH1_GPI_03.PG, 
			iq_stValve := TMO_ROUGH1_VRC_02.iq_stValve)	;
			
IM5K4_PPM_PTM_01(i_xExtIlkOK := IM5K4_PPM_PTM_01_xExtIlkOK, iq_stPTM => );

(*Serial Interface*)
(*Assign adresses to the pfeiffer controllers connected to this serial terminal*)
st_Pfeiffer_CTRL_PTM_Granite2[1].iSerialAddress :=1;//LI3K4_IP1_OUT_PTM_01
st_Pfeiffer_CTRL_PTM_Granite2[1].xEnableComm := TRUE;
st_Pfeiffer_CTRL_PTM_Granite2[2].iSerialAddress :=7;//TM1K4_PTM_01
st_Pfeiffer_CTRL_PTM_Granite2[2].xEnableComm := TRUE;
st_Pfeiffer_CTRL_PTM_Granite2[3].iSerialAddress :=9; //IM5K4_PPM_PTM_01
st_Pfeiffer_CTRL_PTM_Granite2[3].xEnableComm := TRUE;	
(* Instanitate the Function block for serial communication with Pfeiffer*)	
Granite2_PTM_COM(astPfeifferControl := st_Pfeiffer_CTRL_PTM_Granite2,
			   astPfeifferStatus:= st_Pfeiffer_RBK_PTM_Granite2,
				SerialRXBuffer:= K4S6_01_E5_SerialRXBuffer,
				SerialTXBuffer:= K4S6_01_E5_SerialTXBuffer);
(* Copy Status Pv's into the PTM structure*)
LI3K4_IP1_OUT_PTM_01.M_Serial_IO(st_Pfeiffer_CTRL:=st_Pfeiffer_CTRL_PTM_Granite2[1],st_Pfeiffer_RBK:=st_Pfeiffer_RBK_PTM_Granite2[1]);				
TM1K4_PTM_01.M_Serial_IO(st_Pfeiffer_CTRL:=st_Pfeiffer_CTRL_PTM_Granite2[2],st_Pfeiffer_RBK:=st_Pfeiffer_RBK_PTM_Granite2[2]);				
IM5K4_PPM_PTM_01.M_Serial_IO(st_Pfeiffer_CTRL:=st_Pfeiffer_CTRL_PTM_Granite2[3],st_Pfeiffer_RBK:=st_Pfeiffer_RBK_PTM_Granite2[3]);

END_PROGRAM

// ---- POUs/PRG_FSV.TcPOU
PROGRAM PRG_FSV
VAR
END_VAR


TV1K4_VFS_1(
	i_xPMPS_OK:= TRUE, 
	i_xExt_OK:= TRUE, 
	i_sDevName:= 'TV1K4:VFS:01', 
	io_fbFFHWO:= g_FastFaultOutput4 );
	

MR3K4_KBO_VFS_1(
	i_xPMPS_OK:= TRUE, 
	i_xExt_OK:= TRUE, 
	i_sDevName:= 'MR3K4:KBO:VFS:1',
	io_fbFFHWO:= g_FastFaultOutput3
);

MR4K4_KBO_VFS_1(
	i_xPMPS_OK:= TRUE, 
	i_xExt_OK:= TRUE, 
	i_sDevName:= 'MR4K4:KBO:VFS:1',
	io_fbFFHWO:= g_FastFaultOutput3
);
(*FastFaultOuput*)	
g_FastFaultOutput3.Execute(bAutoReset:= TRUE);

END_PROGRAM
